// POUs/Remote/Objects/Basic/[Internal]/FB_BACnetRM_BaseObject
FUNCTION_BLOCK FB_BACnetRM_BaseObject IMPLEMENTS I_BACnetRM_BaseObject
VAR_INPUT CONSTANT
	{region 'Fixed Parameters'}
		{attribute 'parameterCategory':='General'}
		{attribute 'no_copy'}
		Client : REFERENCE TO FB_BACnet_Client;
		{attribute 'parameterCategory':='General'}
		nObjectInstance : UDINT := 16#003FFFFF;	
	{endregion}
END_VAR
VAR
	{region 'Output-Properties'}
		bReady				: BOOL;
	{endregion}
	{region 'SubInit'}
		eObjectType			: E_BACnetObjType				:= 16#FFFF;
		{attribute 'hide'}
		iOwner				: I_BACnetRM_ObjectOwner;												// Owner of current Instance (Pointer to current instance per default)
	{endregion}
END_VAR
VAR
	{region 'General'}
		eErrorID			: E_BACnet_Error				:= E_BACnet_Error.eNoError;
			 
		tObjectID			: T_BACnet_ObjectIdentifier		:= 16#FFFFFFFF;
	{endregion}
END_VAR

IF (NOT bReady) THEN
	IF (iOwner = 0) THEN
		eErrorID := E_BACnet_Error.eInvalidParameter;
		F_BA_LogMessage(ADSLOG_MSGTYPE_ERROR, 'O04', 'Owner of BACnet remote-object not defined!');
		
	ELSIF (__ISVALIDREF(Client)) THEN
		eErrorID := E_BACnet_Error.eNoError;
		bReady := TRUE;
		
		tObjectID := F_BACnet_GetObjId(eObjectType, nObjectInstance);
		
		OnObjectStateChanged();
		
		Client.UpdateRequests();
	ELSE
		eErrorID := E_BACnet_Error.eInvalidClient;
		iOwner.LogMsg.Show(ADSLOG_MSGTYPE_ERROR, 'O17', 'Assigned client-reference is invalid!', FALSE);
	END_IF
ELSE
	// Instance is operational.
END_IF

{attribute 'hide'}
METHOD OnCOV
VAR_INPUT
	ePropID		: E_BACnetPropIdentifier;
END_VAR
// Notify owner:
iOwner.OnBACnetRMObjectCOV(ePropID);
END_METHOD

{attribute 'hide'}
METHOD OnReqError
VAR_INPUT
	iRequest		: I_BACnetRM_Req;
	
	eResult			: E_BACnetRM_Error;
	sLogCode		: STRING			:= '';
END_VAR
VAR
	nLogType		: DWORD;
END_VAR

// (BETA) ... TODO
(*
... eResult ...

eErrorID := ;
nLogType := ADSLOG_MSGTYPE_ERROR;
nLogType := ADSLOG_MSGTYPE_WARN;
*)

iOwner.LogMsg.Show(nLogType, sLogCode, 'TODO: Implement request error!', FALSE);
END_METHOD

METHOD PROTECTED OnObjectStateChanged
// Notify owner:
iOwner.OnBACnetRMObjectStateChanged();
END_METHOD

PROPERTY Error : BOOL
GET
Error := (eErrorID <> E_BACnet_Error.eNoError);
END_GET
END_PROPERTY

PROPERTY ObjectID : T_BACnet_ObjectIdentifier
GET
ObjectID := tObjectID;
END_GET
END_PROPERTY

PROPERTY ObjectInstance : UDINT
GET
ObjectInstance := nObjectInstance;
END_GET
END_PROPERTY

PROPERTY ObjectType : E_BACnetObjType
GET
ObjectType := eObjectType;
END_GET
END_PROPERTY

PROPERTY Ready : BOOL
GET
Ready := bReady;
END_GET
END_PROPERTY

METHOD SyncProperty : BOOL
VAR_INPUT
	ePropID : E_BACnetPropIdentifier;
	nSize : UDINT;
	pData : PVOID;
	eSyncMode : E_BA_SyncModeRM;
END_VAR
CASE (eSyncMode) OF
	E_BA_SyncModeRM.eRead:
		SyncProperty := Client.AddReadProp(ePropID, THIS^, nSize, pData, 16#FFFFFFFF);
	
	E_BA_SyncModeRM.eWrite:
		SyncProperty := Client.AddWriteProp(ePropID, THIS^, nSize, pData, 0, 0, 16);

ELSE
	iOwner.LogMsg.Show1(ADSLOG_MSGTYPE_ERROR, 'SP09', 'Invalid Sync-Mode "%d"!', F_INT(eSyncMode), FALSE);
END_CASE
END_METHOD

METHOD SyncPropertyPrio : BOOL
VAR_INPUT
	ePropID : E_BACnetPropIdentifier;
	nSize : UDINT;
	pData : PVOID;
	pEnable : POINTER TO BOOL := 0;
	pNull : POINTER TO BOOL := 0;
	priority : UDINT := 16;
END_VAR
SyncPropertyPrio := Client.AddWriteProp(ePropID, THIS^, nSize, pData, pEnable, pNull, priority);
END_METHOD

END_FUNCTION_BLOCK

// TEST/TestPackage/CLIENT
PROGRAM CLIENT
VAR
	fbClient			: FB_BACnet_Client					:= (nDeviceInstance := 3637294(*, eReadMode := E_BACnet_CommMode.eCov*));
	
	AV01				: FB_BACnetRM_AV					:= (Client := fbClient, nObjectInstance:=111);
	AVDsp				: FB_BACnetRM_AV_Disp				:= (Client := fbClient, nObjectInstance:=10001);
	AVSp				: FB_BACnetRM_AV_Setp				:= (Client := fbClient, nObjectInstance:=10002);
	AI01				: FB_BACnetRM_AI					:= (Client := fbClient, nObjectInstance:=10000);
	AO01				: FB_BACnetRM_AO					:= (Client := fbClient, nObjectInstance:=10000);
	
	BV01				: FB_BACnetRM_BV					:= (Client := fbClient, nObjectInstance:=99);
	BVDsp				: FB_BACnetRM_BV_Disp				:= (Client := fbClient, nObjectInstance:=10001);
	BVSp				: FB_BACnetRM_BV_Setp				:= (Client := fbClient, nObjectInstance:=10002);
	BI01				: FB_BACnetRM_BI					:= (Client := fbClient, nObjectInstance:=10000);
	BO01				: FB_BACnetRM_BO					:= (Client := fbClient, nObjectInstance:=10000);
	
	MV01				: FB_BACnetRM_MV					:= (Client := fbClient, nObjectInstance:=99);
	MVDsp				: FB_BACnetRM_MV_Disp				:= (Client := fbClient, nObjectInstance:=10001);
	MVSp				: FB_BACnetRM_MV_Setp				:= (Client := fbClient, nObjectInstance:=10002);
	MI01				: FB_BACnetRM_MI					:= (Client := fbClient, nObjectInstance:=10000);
	MO01				: FB_BACnetRM_MO					:= (Client := fbClient, nObjectInstance:=10000);
	
	TLog				: FB_BACnetRM_TLog					:= (Client := fbClient, nObjectInstance:=10000);
	TLM					: FB_BACnetRM_TLM					:= (Client := fbClient, nObjectInstance:=10000);
	Cal01				: FB_BACnetRM_Cal					:= (Client := fbClient, nObjectInstance:=10000);
	SchedA				: FB_BACnetRM_SchedA				:= (Client := fbClient, nObjectInstance:=10000);
	SchedB				: FB_BACnetRM_SchedB				:= (Client := fbClient, nObjectInstance:=10001);
	SchedM				: FB_BACnetRM_SchedM				:= (Client := fbClient, nObjectInstance:=10002);
	Loop1				: FB_BACnetRM_Loop					:= (Client := fbClient, nObjectInstance:=10000);
	Loop2				: FB_BACnetRM_CnvLoop				:= (Client := fbClient, nObjectInstance:=10000);
	
	NC_AlmStd			: FB_BACnetRM_NC					:= (Client := fbClient, nObjectInstance:=11);
	
	Acc					: FB_BACnetRM_Acc					:= (Client := fbClient, nObjectInstance:=10000);
	PC					: FB_BACnetRM_PC					:= (Client := fbClient, nObjectInstance:=10000);
	Prog				: FB_BACnetRM_Prog					:= (Client := fbClient, nObjectInstance:=10000);
END_VAR
VAR
	diag : ST_BACnet_Diagnosis;
	scanRes : ARRAY [0..99] OF ST_BACnetRM_ScanResult;
	syncTime : ST_BA_DateTime;
	
	bDiag : BOOL;
	bScan : BOOL;
	bGet : BOOL;
	bSync : BOOL;
END_VAR

fbClient();

AV01();
AVDsp();
AVSp();
AI01();
AO01();

BV01();
BVDsp();
BVSp();
BI01();
BO01();

MV01();
MVDsp();
MVSp();
MI01();
MO01();

TLog();
TLM();
Cal01();
SchedA();
SchedB();
SchedM();
Loop1();
Loop2();

NC_AlmStd();

Acc();
PC();
Prog();

IF bDiag THEN
	fbClient.Adapter.GetDiagnosis(ADR(diag));
END_IF

IF bScan THEN	
	fbClient.Adapter.StartScan();
	bScan:=FALSE;
END_IF

IF bGet THEN
	fbClient.Adapter.GetScanResult(ADR(scanRes), 100);
	bGet:=FALSE;
END_IF

IF bSync THEN
	fbClient.Adapter.TimeSync(ADR(syncTime), TRUE);
	bSync:=FALSE;
END_IF

END_PROGRAM

// POUs/Remote/FB_BACnet_Client
FUNCTION_BLOCK FB_BACnet_Client IMPLEMENTS I_BACnetRM_Object
VAR_INPUT CONSTANT
	{region 'Fixed Parameters'}
		{attribute 'parameterCategory':='General'}
		{attribute 'no_copy'}
		Adapter	: REFERENCE TO FB_BACnet_Adapter := BACnet_Globals.DefaultAdapter;
		{attribute 'parameterCategory':='General'}
		nDeviceInstance : UDINT;
	{endregion}
END_VAR
VAR_INPUT CONSTANT PERSISTENT
	{region 'Variable Parameters'}
		{attribute 'parameterCategory':='Communication'}
		nMaxParallelRequests : UDINT := 1;
		{attribute 'parameterCategory':='Communication'}
		nRPMPropertiesPerRequest : UDINT := 80;
		{attribute 'parameterCategory':='Communication'}
		tCOVLifeTime : TIME := T#300S;	
		{attribute 'parameterCategory':='Communication'}
		eReadMode : E_BACnet_CommMode;
		{attribute 'parameterCategory':='Communication'}
		tReadCycleTime : TIME := T#5S;
		{attribute 'parameterCategory':='Communication'}
		tWriteCycleTime : TIME := T#5S;
	{endregion}
END_VAR
VAR_OUTPUT
	bReady					: BOOL;
	eErrorID				: E_BACnet_Error;
	nAdsPort 				: UINT;
	bConnected  			: BOOL;
END_VAR
VAR
	{region 'General'}
		tObjectID			: T_BACnet_ObjectIdentifier		:= 16#FFFFFFFF;
	{endregion}
END_VAR
VAR
	{region 'General'}
		eState				: E_BACnetRM_ClientState;
	
		stSupportedServices	: ST_BACnet_ServicesSupportedBits;
	{endregion}
	{region 'Request Lists'}
		{region 'Read'}
			{attribute 'hide'}
			stReadList 		: POINTER TO ST_BACnetRM_ReadEntry;
			{attribute 'hide'}
			nReadList		: UDINT := 0;
			{attribute 'hide'}
			nReadMax		: UDINT := 0;
		{endregion}
		{region 'Write'}
			{attribute 'hide'}
			stWriteList		: POINTER TO ST_BACnetRM_WriteEntry;
			{attribute 'hide'}
			nWriteList		: UDINT := 0;
			{attribute 'hide'}
			nWriteMax		: UDINT := 0;	
		{endregion}
	{endregion}
	{region 'Request Fifo'}
		{region 'Cyclic'}
			{attribute 'hide'}
			stReqList		: POINTER TO ST_BACnetRM_ReqPtr := 0;
			{attribute 'hide'}
			nReqList		: UDINT := 0;
			{attribute 'hide'}
			nCurReq			: UDINT := 0;
		{endregion}
		{region 'Acyclic / Dynamic'}
			{attribute 'hide'}
			fbReadFifo		: FB_BACnetRM_ReqFifo := (Client := THIS^);
			{attribute 'hide'}
			fbWriteFifo		: FB_BACnetRM_ReqFifo := (Client := THIS^);
		{endregion}
				  
		nOpenReq			: UDINT := 0;
		{attribute 'hide'}
		bUpdateReqs			: BOOL;
	{endregion}
		 
	{region 'Internal'}
		{attribute 'hide'}
		iServer				: ITcIoBACnetPlcServer;
		{attribute 'hide'}
		iClient				: ITcIoBACnetPlcClient;
		{attribute 'hide'}
		iDevice				: ITcIoBACnetPlcDevice;
		{attribute 'hide'}
		_bCreated			: BOOL;
		{attribute 'hide'}
		nUpdateCountAdp		: UDINT := 0;
			 
		{attribute 'hide'}
		fbRead				: FB_BACnetRM_ReadProperty := (Client:=THIS^);
		{attribute 'hide'}
		_ClientStatus		: WORD;
		{attribute 'hide'}
		_ClientControl		: WORD;
	{endregion}
END_VAR
VAR_TEMP
	n						: UDINT := 0;
END_VAR

IF __ISVALIDREF(Adapter) THEN
	IF Adapter._nUpdateCount = nUpdateCountAdp THEN
		Adapter();
	END_IF
	(* remind current number of update counter *)
	nUpdateCountAdp := Adapter._nUpdateCount;
	
	IF iDevice = 0 THEN
		iDevice := Adapter.Device;
	END_IF
END_IF

IF iClient = 0 THEN
	IF iDevice <> 0 THEN
		IF S_OK <> iDevice.GetClientById(nDeviceInstance, ADR(iServer)) THEN
			IF NOT _bCreated THEN
				IF S_OK = iDevice.CreateClient(nDeviceInstance) THEN
					_bCreated := TRUE;
				END_IF
			END_IF			
		ELSE
			iServer.GetAdsPort(ADR(nAdsPort));
			IF S_OK <> iServer.TcQueryInterface(TC_GLOBAL_IID_LIST.IID_ITcIoBACnetPlcClient, ADR(iClient)) THEN
				eErrorID := E_BACnet_Error.eInvalidClient;
			END_IF
		END_IF
	END_IF
END_IF

IF iClient <> 0 THEN
	iServer.UpdateDeviceStatus(ADR(_ClientControl), ADR(_ClientStatus));	
	IF Adapter.bEthernetLink THEN
		bConnected := NOT (SHR((_ClientStatus AND 16#FF00), 8) < 4);
	ELSE
		bConnected := FALSE;
	END_IF
	CASE eState OF
		E_BACnetRM_ClientState.eInit:
			IF bConnected THEN
				tObjectID := F_BACnet_GetObjId(ObjectType, nDeviceInstance);
		
				IF stSupportedServices.bSuppReadProperty THEN
					eState:=E_BACnetRM_ClientState.eCalcAuto;
				ELSE
					eState:=E_BACnetRM_ClientState.eReadSupportedServices;
				END_IF
			END_IF
		E_BACnetRM_ClientState.eReadSupportedServices:
			IF fbRead.bReady THEN
				IF eReadMode = E_BACnet_CommMode.eAuto OR eReadMode = E_BACnet_CommMode.eRpm THEN
					fbReadFifo.bRpm:=stSupportedServices.bSuppReadPropertyMultiple;
				END_IF
				eState:=E_BACnetRM_ClientState.eCalcAuto;
			ELSIF fbRead.bError THEN
				eState:=E_BACnetRM_ClientState.eError;
			ELSIF NOT fbRead.bBusy THEN
				fbRead(iObject:=THIS^, ePropID:=E_BACnetPropIdentifier.PropProtocolServicesSupported, nData:=SIZEOF(stSupportedServices), pData:=ADR(stSupportedServices), bExecute:=TRUE);
			END_IF
			fbReadFifo.ProcessReadFifo();
		E_BACnetRM_ClientState.eCalcAuto:
			IF nReadList > 0 OR nWriteList>0 THEN
				IF eReadMode = E_BACnet_CommMode.eAuto THEN
					IF nReadList > 300 AND stSupportedServices.bSuppReadPropertyMultiple THEN
						eReadMode := E_BACnet_CommMode.eRpm;
					ELSIF stSupportedServices.bSuppSubscribeCOV THEN
						eReadMode := E_BACnet_CommMode.eCov;
					ELSIF stSupportedServices.bSuppReadPropertyMultiple THEN
						eReadMode := E_BACnet_CommMode.eRpm;
					ELSE
						eReadMode := E_BACnet_CommMode.eRp;
					END_IF
				END_IF
				eState:=E_BACnetRM_ClientState.eCreateRequests;
			ELSE
				eState:=E_BACnetRM_ClientState.eCycle;
			END_IF
			eState:=E_BACnetRM_ClientState.eCreateRequests;
		E_BACnetRM_ClientState.eCreateRequests:
			IF CreateReqList() THEN
				bUpdateReqs := FALSE;
				eState:=E_BACnetRM_ClientState.eCycle;
			END_IF
		E_BACnetRM_ClientState.eCycle:
			IF bUpdateReqs THEN
				eState:=E_BACnetRM_ClientState.eReInit;
				bUpdateReqs := FALSE;
			ELSE
				bReady:=TRUE;
				
				// Work on acyclic / dynamic requests:
				fbReadFifo.ProcessReadFifo();
				fbWriteFifo.ProcessWriteFifo();
				
				// Work on cyclic requests:
				IF stReqList <> 0 THEN
					WHILE nOpenReq < nMaxParallelRequests AND n<nReqList DO								
						IF stReqList[nCurReq].pPtr <> 0 AND_THEN stReqList[nCurReq].fbBase^.IsReady() THEN
							IF stReqList[nCurReq].fbBase^.Send() THEN
								nOpenReq:=nOpenReq+1;
							END_IF
						END_IF
						n:=n+1;
						nCurReq:=(nCurReq+1) MOD nReqList;
					END_WHILE
				END_IF
			END_IF
			IF NOT bConnected THEN
				eState:=E_BACnetRM_ClientState.eReInit;
			END_IF
		E_BACnetRM_ClientState.eReInit:
			DeleteReqList();
			eState:=E_BACnetRM_ClientState.eInit;
		E_BACnetRM_ClientState.eError:
			// Todo: add 5 sec timer 
			eState:=E_BACnetRM_ClientState.eReInit;
	END_CASE
END_IF

{attribute 'hide'}
METHOD OnCOV
VAR_INPUT
	ePropID		: E_BACnetPropIdentifier;
END_VAR
END_METHOD

{attribute 'hide'}
METHOD OnReqError
VAR_INPUT
	iRequest		: I_BACnetRM_Req;
	
	eResult			: E_BACnetRM_Error;
	sLogCode		: STRING			:= '';
END_VAR
VAR
	nLogType		: DWORD;
END_VAR
END_METHOD

METHOD INTERNAL OnRequestComplete
IF nOpenReq > 0 THEN
	nOpenReq:=nOpenReq-1;
END_IF
END_METHOD

METHOD INTERNAL AddFifoReadReq : BOOL
VAR_INPUT
	pReq : POINTER TO FB_BACnetRM_ReadProperty;
END_VAR
VAR
	entry : ST_BACnetRM_FifoEntry;
END_VAR
entry.fbRead:=pReq;
AddFifoReadReq:=fbReadFifo.AddFifoReq(entry);
END_METHOD

METHOD INTERNAL AddFifoWriteReq : BOOL
VAR_INPUT
	pReq : POINTER TO FB_BACnetRM_WriteProperty;
END_VAR
VAR
	entry : ST_BACnetRM_FifoEntry;
END_VAR
entry.fbWrite:=pReq;
AddFifoWriteReq:=fbWriteFifo.AddFifoReq(entry);
END_METHOD

METHOD INTERNAL UpdateRequests 
VAR_INPUT
END_VAR
bUpdateReqs:=TRUE;
END_METHOD

METHOD PRIVATE CreateReadReq : I_BACnetRM_Req
VAR_INPUT
	eReadMode : E_BACnet_CommMode;
	stEntry : ST_BACnetRM_ReadEntry;
END_VAR
VAR
	stPtr : ST_BACnetRM_ReqPtr;
END_VAR
CASE eReadMode OF
	E_BACnet_CommMode.eCov:
		stPtr.fbCov:=__NEW(FB_BACnetRM_ReqCov);
		IF stPtr.fbCov <> 0 THEN
			stPtr.fbCov^(Client:=THIS^,iObject:=stEntry.iObject,  ePropID:=stEntry.ePropID, tLifetime:=tCOVLifeTime, pData:=stEntry.pData, nData:=stEntry.nData);
			stPtr.fbCov^.InitTimer();
		END_IF
		CreateReadReq:=stPtr.iReq;
		RETURN;
	E_BACnet_CommMode.eCovC:
		stPtr.fbCov:=__NEW(FB_BACnetRM_ReqCov);
		IF stPtr.fbCov <> 0 THEN
			stPtr.fbCov^(Client:=THIS^,iObject:=stEntry.iObject, bConfirmed:=TRUE, ePropID:=stEntry.ePropID, tLifetime:=tCOVLifeTime, pData:=stEntry.pData, nData:=stEntry.nData);
			stPtr.fbCov^.InitTimer();
		END_IF
		CreateReadReq:=stPtr.iReq;
		RETURN;
	E_BACnet_CommMode.eCovU:
		stPtr.fbCov:=__NEW(FB_BACnetRM_ReqCov);
		IF stPtr.fbCov <> 0 THEN
			stPtr.fbCov^(Client:=THIS^,iObject:=stEntry.iObject, bUnsubscribed:=TRUE, ePropID:=stEntry.ePropID, tLifetime:=tCOVLifeTime, pData:=stEntry.pData, nData:=stEntry.nData);
			stPtr.fbCov^.InitTimer();
		END_IF
		CreateReadReq:=stPtr.iReq;
		RETURN;
	E_BACnet_CommMode.eRp:
		stPtr.fbRead:=__NEW(FB_BACnetRM_ReqRead);
		IF stPtr.fbRead <> 0 THEN
			stPtr.fbRead^(Client:=THIS^,iObject:=stEntry.iObject, tCycleTime:=tReadCycleTime, ePropID:=stEntry.ePropID, pData:=stEntry.pData, nData:=stEntry.nData);
			stPtr.fbRead^.InitTimer();
		END_IF
		CreateReadReq:=stPtr.iReq;
		RETURN;
	E_BACnet_CommMode.eRpm:
		stPtr.fbRpm:=__NEW(FB_BACnetRM_ReqRpm);
		IF stPtr.fbRpm <> 0 THEN
			stPtr.fbRpm^(Client:=THIS^,iObject:=stEntry.iObject, tCycleTime:=tReadCycleTime);
			stPtr.fbRpm^.InitTimer();
		END_IF
		CreateReadReq:=stPtr.iReq;
		RETURN;
END_CASE
END_METHOD

METHOD PRIVATE CreateReqList : BOOL
VAR_INPUT
END_VAR
VAR
	i : UDINT;
	nReqs : UDINT;
	stPtr : ST_BACnetRM_ReqPtr;
	nReqsLeft : UDINT;
END_VAR
DeleteReqList();

IF eReadMode = E_BACnet_CommMode.eRpm THEN
	nReqs:=((nReadList+nRPMPropertiesPerRequest-1)/nRPMPropertiesPerRequest);
ELSE
	nReqs := nReadList;
END_IF

nReqs:=nReqs+nWriteList;

IF nReqs = 0 THEN
	RETURN;
END_IF

stReqList:=__NEW(POINTER TO ST_BACnetRM_ReqPtr, nReqs);

IF stReqList = 0 THEN
	RETURN;
END_IF

IF eReadMode = E_BACnet_CommMode.eRpm THEN
	nReqsLeft:=nReadList;
	WHILE nReqsLeft > 0 DO
		 stPtr.fbRpm:=__NEW(FB_BACnetRM_ReqRpm);
		 IF stPtr.fbRpm = 0 THEN
			 RETURN;
		 END_IF
		 stPtr.fbRpm^(Client:=THIS^, iObject:=stReadList[i].iObject, tCycleTime:=tReadCycleTime, pEntries:=ADR(stReadList[i]), nEntries:=MIN(nRPMPropertiesPerRequest, nReqsLeft));
		 stPtr.fbRpm^.InitTimer();
		 stPtr.fbRpm^.UpdateRequest();
		 nReqsLeft:=MIN(0, nReqsLeft-nRPMPropertiesPerRequest);
		 stReqList[nReqList]:=stPtr;
		 i:=i+MIN(0, nReqsLeft-nRPMPropertiesPerRequest);
		 nReqList:=nReqList+1;
	END_WHILE
	
ELSIF (nReadList > 0) THEN
	FOR i:=0 TO nReadList-1 DO
		stReqList[nReqList].iReq := CreateReadReq(eReadMode, stReadList[i]);
		IF stReqList[nReqList].pPtr = 0 THEN
			RETURN;
		END_IF
		nReqList:=nReqList+1;
	END_FOR
END_IF

IF eReadMode = E_BACnet_CommMode.eCov OR eReadMode = E_BACnet_CommMode.eCovC OR eReadMode = E_BACnet_CommMode.eCovU THEN
	OptimizeCOV();
END_IF

IF (nWriteList > 0) THEN
	FOR i:=0 TO nWriteList-1 DO
		stReqList[nReqList].fbWrite := __NEW(FB_BACnetRM_ReqWrite);
		IF stReqList[nReqList].pPtr = 0 THEN
			RETURN;
		END_IF
		
		stReqList[nReqList].fbWrite^(Client:=THIS^, iObject:=stWriteList[i].iObject, ePropID:=stWriteList[i].ePropID, tCycleTime:=tWriteCycleTime, pData:=stWriteList[i].pData, nData:=stWriteList[i].nData, pEnable:=stWriteList[i].pEnable, pNull:=stWriteList[i].pNull, fCOVIncrement:=stWriteList[i].fCOVIncrement, nPriority:=stWriteList[i].nPriority);
		stReqList[nReqList].fbWrite^.InitTimer();
		nReqList:=nReqList+1;
	END_FOR
END_IF

nCurReq := 0;
nOpenReq := 0;
CreateReqList:=TRUE;
END_METHOD

METHOD PRIVATE DeleteReqList
VAR_INPUT
END_VAR
VAR
	i : UDINT;
END_VAR
IF nReqList > 0 AND stReqList <> 0 THEN
	FOR i:=0 TO nReqList-1 DO
		IF stReqList[i].nByte <> 0 THEN
			CASE stReqList[i].iReq.GetRequestType() OF
				E_BACnetRM_RequestType.eRead:__DELETE(stReqList[i].fbRead);
				E_BACnetRM_RequestType.eReadPropertyMultiple:__DELETE(stReqList[i].fbRpm); 
				E_BACnetRM_RequestType.eWrite:__DELETE(stReqList[i].fbWrite);
				E_BACnetRM_RequestType.eWritePropertyMultiple:__DELETE(stReqList[i].fbWpm);
				E_BACnetRM_RequestType.eCOV_C:__DELETE(stReqList[i].fbCov);
				E_BACnetRM_RequestType.eCOV:__DELETE(stReqList[i].fbCov);
				E_BACnetRM_RequestType.eCOV_U:__DELETE(stReqList[i].fbCov);
			END_CASE
		END_IF
	END_FOR
	__DELETE(stReqList);
	stReqList:=0;
	nReqList:=0;
END_IF
END_METHOD

// Optimizes request count per object.
// > If a single object has more than one request, these multiple requests can be handled via a single RPM-request.
METHOD PRIVATE OptimizeCOV : BOOL
VAR
	i : UDINT;
	j : UDINT;
END_VAR
IF (nReadList > 0) THEN
	FOR i:=0 TO nReadList-1 DO
		IF stReqList[i].fbCov^.Master = 0 THEN
			FOR j:=i+1 TO nReadList-1 DO
				IF stReqList[i].fbCov^.iObject = stReqList[j].fbCov^.iObject THEN
					 stReqList[i].fbCov^.AddCovSlave(stReqList[j].fbCov);
					 stReqList[j].fbCov^.Master:=stReqList[i].fbCov;
					 IF stReqList[i].fbCov^.fCOVIncrement = 0 AND stReqList[i].fbCov^.ePropID = E_BACnetPropIdentifier.PropPresentValue AND stReqList[j].fbCov^.ePropID = E_BACnetPropIdentifier.PropStatusFlags THEN
						  stReqList[j].fbCov^.SendSubscription:=FALSE;
					 END_IF
				END_IF
			END_FOR
		END_IF
	END_FOR
END_IF
END_METHOD

// Called after online change.
{attribute 'call_after_online_change_slot' := '10'}
METHOD PROTECTED OnPostOnlineChange
IF iServer <> 0 THEN
	FW_SafeRelease(ADR(iServer));
	iServer:=0;
END_IF
IF iClient <> 0 THEN
	FW_SafeRelease(ADR(iClient));
	iClient:=0;
END_IF
iDevice:=0;

eState:=E_BACnetRM_ClientState.eReInit;
END_METHOD

METHOD FB_Exit : BOOL
VAR_INPUT
	 bInCopyCode : BOOL; // if TRUE, the exit method is called for exiting an instance that is copied afterwards (online change).
END_VAR
IF iServer <> 0 THEN
	iServer.OnPlcAction(E_BACnet_PlcAction.eSuspend);
	iServer:=0;
END_IF
IF iClient <> 0 THEN
	FW_SafeRelease(ADR(iClient));
	iClient:=0;
END_IF

iDevice:=0;

DeleteReqList();

IF stReadList <> 0 THEN
	__DELETE(stReadList);
	stReadList:=0;
END_IF
IF stWriteList <> 0 THEN
	__DELETE(stWriteList);
	stWriteList:=0;
END_IF
END_METHOD

PROPERTY Error : BOOL
GET
Error := (eErrorID <> E_BACnet_Error.eNoError);
END_GET
END_PROPERTY

PROPERTY ObjectID : T_BACnet_ObjectIdentifier
GET
ObjectID := tObjectID;
END_GET
END_PROPERTY

PROPERTY ObjectInstance : UDINT
GET
ObjectInstance := nDeviceInstance;
END_GET
END_PROPERTY

PROPERTY ObjectType : E_BACnetObjType
GET
ObjectType := E_BACnetObjType.ObjDevice;
END_GET
END_PROPERTY

PROPERTY OpenRequestCount : UDINT
GET
OpenRequestCount:=nOpenReq;
END_GET
SET
nOpenReq:=OpenRequestCount;
END_SET
END_PROPERTY

PROPERTY Ready : BOOL
GET
Ready := bReady;
END_GET
END_PROPERTY

METHOD AddReadProp : BOOL
VAR_INPUT
	ePropID : E_BACnetPropIdentifier;
	iObject : I_BACnetRM_BaseObject;
	nData : UDINT;
	pData : PVOID;
	nIndex : UDINT := 16#FFFFFFFF;
END_VAR
VAR
	nTmp : UDINT;
	nTmpSize : UDINT;
	pTmp : PVOID;
END_VAR
IF nReadList+1 >= nReadMax THEN
	nTmp := nReadMax+10;
	nTmpSize := nTmp*SIZEOF(ST_BACnetRM_ReadEntry);
	pTmp := __NEW(BYTE,nTmpSize);
	IF pTmp = 0 THEN
		RETURN;
	END_IF
	IF stReadList <> 0 THEN
		MEMCPY(pTmp, stReadList, nReadMax*SIZEOF(ST_BACnetRM_ReadEntry));
		__DELETE(stReadList);
	END_IF
	stReadList:=pTmp;
	nReadMax:=nTmp;
END_IF

MEMSET(ADR(stReadList[nReadList]), 0, SIZEOF(ST_BACnetRM_ReadEntry));

stReadList[nReadList].iObject:=iObject;
stReadList[nReadList].ePropID:=ePropID;
stReadList[nReadList].pData:=pData;
stReadList[nReadList].nData:=nData;
stReadList[nReadList].nIndex:=nIndex;

nReadList := nReadList + 1;

AddReadProp:=TRUE;
END_METHOD

METHOD AddWriteProp : BOOL
VAR_INPUT
	ePropID : E_BACnetPropIdentifier;
	iObject : I_BACnetRM_BaseObject;
	nData : UDINT;
	pData : PVOID;
	pEnable : POINTER TO BOOL := 0;
	pNull : POINTER TO BOOL := 0;
	nPriority : UDINT := 16;
END_VAR
VAR
	nTmp : UDINT;
	nTmpSize : UDINT;
	pTmp : PVOID;
END_VAR
IF nWriteList+1 >= nWriteMax THEN
	nTmp := nWriteMax+10;
	nTmpSize := nTmp*SIZEOF(ST_BACnetRM_WriteEntry);
	pTmp := __NEW(BYTE,nTmpSize);
	IF pTmp = 0 THEN
		RETURN;
	END_IF
	IF stWriteList <> 0 THEN
		MEMCPY(pTmp, stWriteList, nWriteMax*SIZEOF(ST_BACnetRM_WriteEntry));
		__DELETE(stWriteList);
	END_IF
	stWriteList:=pTmp;
	nWriteMax:=nTmp;
END_IF

MEMSET(ADR(stWriteList[nWriteList]), 0, SIZEOF(ST_BACnetRM_WriteEntry));

stWriteList[nWriteList].iObject:=iObject;
stWriteList[nWriteList].ePropID:=ePropID;
stWriteList[nWriteList].pData:=pData;
stWriteList[nWriteList].nData:=nData;
stWriteList[nWriteList].nPriority:=nPriority;
stWriteList[nWriteList].pEnable:=pEnable;
stWriteList[nWriteList].pNull:=pNull;
stWriteList[nWriteList].fCOVIncrement := 0.0;

nWriteList := nWriteList + 1;

AddWriteProp:=TRUE;
END_METHOD

END_FUNCTION_BLOCK

// POUs/Remote/Requests/[Internal]/FB_BACnetRM_ReqFifo
{attribute 'c++_compatible'}
{attribute 'enable_dynamic_creation'}
{attribute 'hide'}
FUNCTION_BLOCK FB_BACnetRM_ReqFifo EXTENDS FB_BACnetRM_ReqBase
VAR_INPUT
	bRpm : BOOL;
	bWpm : BOOL;
END_VAR
VAR
	pReqFifo	: POINTER TO ST_BACnetRM_FifoEntry;
	nReqFifo	: UDINT := 0;
	nMaxFifo	: UDINT := 0;
	nPendFifo	: UDINT := 0;
END_VAR

METHOD INTERNAL AddFifoReq : BOOL
VAR_INPUT
	pEntry : ST_BACnetRM_FifoEntry;
END_VAR
VAR
	nTmp : UDINT;
	nTmpSize : UDINT;
	pTmp : POINTER TO ST_BACnetRM_FifoEntry;
END_VAR
IF nReqFifo+1 >= nMaxFifo THEN
	nTmp := 2*nMaxFifo+100;
	nTmpSize := nTmp*SIZEOF(ST_BACnetRM_FifoEntry);
	pTmp := __NEW(BYTE,nTmpSize);
	IF pTmp = 0 THEN
		RETURN;
	END_IF
	IF pReqFifo <> 0 THEN
		MEMCPY(pTmp, pReqFifo, nMaxFifo*SIZEOF(ST_BACnetRM_FifoEntry));
		__DELETE(pReqFifo);
	END_IF
	pReqFifo:=pTmp;
	nMaxFifo:=nTmp;
END_IF

pReqFifo[nReqFifo]:=pEntry;
nReqFifo:=nReqFifo+1;

AddFifoReq:=TRUE;
END_METHOD

METHOD INTERNAL ProcessReadFifo : BOOL
VAR_INPUT
END_VAR
VAR
	pRequest : ST_BACnetRM_ReqPtr;
	nSize : UDINT;
	n :UDINT;
	pEntries : POINTER TO ST_BACnetRM_ReadEntry;
	
	x : UDINT;
END_VAR
IF IsValid THEN
	WHILE Client.nOpenReq < Client.nMaxParallelRequests AND nReqFifo > 0 DO		
		IF bRpm AND nReqFifo>1 THEN
			n:=0;
			nSize:=MIN(nReqFifo, Client.nRPMPropertiesPerRequest)*SIZEOF(ST_BACnetRM_ReadEntry);
			pRequest.fbRpm := __NEW(FB_BACnetRM_ReqRpm);
			IF pRequest.fbRpm = 0 THEN
				RETURN;
			END_IF
			pEntries:=__NEW(BYTE,nSize);
			IF pEntries = 0 THEN
				__DELETE(pRequest.fbRpm);
				RETURN;
			END_IF
			WHILE n<nReqFifo AND n < Client.nRPMPropertiesPerRequest DO
				pEntries[n].iObject:=pReqFifo[n].fbRead^.iObject;
				pEntries[n].ePropID:=pReqFifo[n].fbRead^.ePropID;
				pEntries[n].pData:=pReqFifo[n].fbRead^.pData;
				pEntries[n].nData:=pReqFifo[n].fbRead^.nData;
				pEntries[n].nIndex:=pReqFifo[n].fbRead^.nIndex;
				pEntries[n].fbReadProp:=pReqFifo[n].fbRead;
				n:=n+1;
			END_WHILE		
			pRequest.fbRpm^(Client:=Client, pEntries:=pEntries, nEntries:=n, bFreeEntries:=TRUE);
			IF pRequest.fbRpm^.UpdateRequest() AND_THEN pRequest.fbRpm^.Send() THEN
				Client.OpenRequestCount:=Client.nOpenReq+1;
				pReqFifo[0].fbRead^.Request:=pRequest;
				pReqFifo[0].fbRead^.bRequestRPM:=TRUE;
				MEMMOVE(pReqFifo, ADR(pReqFifo[n]), n*SIZEOF(ST_BACnetRM_ReadEntry));
				nReqFifo:=nReqFifo-n;
			ELSE
				__DELETE(pRequest.fbRpm);
				RETURN;
			END_IF
		ELSE
			pRequest.fbRead := __NEW(FB_BACnetRM_ReqRead);
			IF pRequest.fbRead = 0 THEN
				RETURN;
			END_IF
			pRequest.fbRead^(Client:=Client, iObject:=pReqFifo[0].fbRead^.iObject, pData:=pReqFifo[0].fbRead^.pData, nData:=pReqFifo[0].fbRead^.nData, ePropID:=pReqFifo[0].fbRead^.ePropID, fbReadProp:=pReqFifo[0].fbRead);
			IF pRequest.fbRead^.Send() THEN
				Client.OpenRequestCount:=Client.nOpenReq+1;
				pReqFifo[0].fbRead^.Request:=pRequest;	
				pReqFifo[0].fbRead^.bRequestRPM:=FALSE;
				MEMMOVE(pReqFifo, ADR(pReqFifo[1]), 1*SIZEOF(ST_BACnetRM_ReadEntry));
				nReqFifo:=nReqFifo-1;
			ELSE
				__DELETE(pRequest.fbRead);
				RETURN;
			END_IF
		END_IF
	END_WHILE
	
	ProcessReadFifo:=TRUE;
ELSE
	// (BETA) ... Output Error
END_IF
END_METHOD

METHOD INTERNAL ProcessWriteFifo : BOOL
VAR_INPUT
END_VAR
VAR
	pRequest : ST_BACnetRM_ReqPtr;
	nSize : UDINT;
	n :UDINT;
	pEntries : POINTER TO ST_BACnetRM_ReadEntry;
END_VAR
IF IsValid THEN
	WHILE Client.nOpenReq < Client.nMaxParallelRequests AND nReqFifo > 0 DO		
		IF bWpm THEN
			n:=0;
			nSize:=MIN(nReqFifo, Client.nRPMPropertiesPerRequest)*SIZEOF(ST_BACnetRM_ReadEntry);
			pRequest.fbWpm:= __NEW(FB_BACnetRM_ReqWpm);
			IF pRequest.fbWpm = 0 THEN
				RETURN;
			END_IF
			pEntries:=__NEW(BYTE,nSize);
			IF pEntries = 0 THEN
				__DELETE(pRequest.fbWpm);
				RETURN;
			END_IF
			WHILE n<nReqFifo-1 AND n < Client.nRPMPropertiesPerRequest DO
				pEntries[n].iObject:=pReqFifo[n].fbWrite^.iObject;
				pEntries[n].ePropID:=pReqFifo[n].fbWrite^.ePropID;
				pEntries[n].pData:=pReqFifo[n].fbWrite^.pData;
				pEntries[n].nData:=pReqFifo[n].fbWrite^.nData;
				pEntries[n].nIndex:=pReqFifo[n].fbWrite^.nIndex;
				pEntries[n].fbReadProp:=pReqFifo[n].fbWrite;
				n:=n+1;
			END_WHILE
			pRequest.fbWpm^(Client:=Client, pEntries:=pEntries, nEntries:=n, bFreeEntries:=TRUE);
			IF pRequest.fbWpm^.UpdateRequest() AND_THEN pRequest.fbWpm^.Send() THEN
				Client.OpenRequestCount:=Client.nOpenReq+1;
				pReqFifo[0].fbRead^.Request:=pRequest;
				pReqFifo[0].fbWrite^.bRequestWPM:=TRUE;
				MEMMOVE(pReqFifo, ADR(pReqFifo[n]), n*SIZEOF(ST_BACnetRM_ReadEntry));
				nReqFifo:=nReqFifo-n;
			ELSE
				__DELETE(pRequest.fbWpm);
				RETURN;
			END_IF
		ELSE
			pRequest.fbWrite := __NEW(FB_BACnetRM_ReqWrite);
			IF pRequest.fbWrite = 0 THEN
				RETURN;
			END_IF
			pRequest.fbWrite^(Client:=Client, iObject:=pReqFifo[0].fbWrite^.iObject, ePropID:=pReqFifo[0].fbWrite^.ePropID, pData:=pReqFifo[0].fbWrite^.pData, nData:=pReqFifo[0].fbWrite^.nData, fbWriteProp:=pReqFifo[0].fbWrite);
			IF pRequest.fbWrite^.Send() THEN
				pReqFifo[0].fbWrite^.Request:=pRequest;	
				pReqFifo[0].fbWrite^.bRequestWPM:=FALSE;
				Client.OpenRequestCount:=Client.nOpenReq+1;
				MEMMOVE(pReqFifo, ADR(pReqFifo[1]), 1*SIZEOF(ST_BACnetRM_ReadEntry));
			ELSE
				__DELETE(pRequest.fbWrite);
				RETURN;
			END_IF
		END_IF
	END_WHILE
	
	ProcessWriteFifo:=TRUE;
ELSE
	// (BETA) ... Output Error
END_IF
END_METHOD

METHOD FB_Exit : BOOL
VAR_INPUT
	 bInCopyCode : BOOL; // if TRUE, the exit method is called for exiting an instance that is copied afterwards (online change).
END_VAR
IF pReqFifo <> 0 THEN
	__DELETE(pReqFifo);
	pReqFifo:=0;
END_IF
END_METHOD

PROPERTY IsValid : BOOL
GET
// Hint:
// > Don't call "super()"!
//   The "iObject" Interface-pointer is ignored to this instance because it is unused.
IsValid := (__ISVALIDREF(Client));
END_GET
END_PROPERTY

END_FUNCTION_BLOCK

// POUs/Remote/Requests/[Internal]/[Base]/FB_BACnetRM_ReqBase
{attribute 'c++_compatible'}
{attribute 'enable_dynamic_creation'}
{attribute 'hide'}
FUNCTION_BLOCK FB_BACnetRM_ReqBase IMPLEMENTS I_BACnetRM_Req
VAR_INPUT
	{attribute 'initialize_on_call'}
	{attribute 'no_copy'}
	Client : REFERENCE TO FB_BACnet_Client;
	iObject : I_BACnetRM_BaseObject;
END_VAR

METHOD GetRequestType : E_BACnetRM_RequestType
VAR_INPUT
END_VAR
GetRequestType:=E_BACnetRM_RequestType.eUndefined;
END_METHOD

METHOD IsReady : BOOL
VAR_INPUT
END_VAR
END_METHOD

PROPERTY IsValid : BOOL
GET
VAR
	iTest : BOOL;
END_VAR
IsValid := (__ISVALIDREF(Client)) AND (iObject <> 0);
END_GET
END_PROPERTY

METHOD Send : BOOL
VAR
	_ClTmp : ITcIoBACnetPlcClient;
END_VAR
END_METHOD

END_FUNCTION_BLOCK

// POUs/Remote/Requests/[Internal]/FB_BACnetRM_ReqRpm
{attribute 'c++_compatible'}
{attribute 'enable_dynamic_creation'}
{attribute 'hide'}
FUNCTION_BLOCK FB_BACnetRM_ReqRpm EXTENDS FB_BACnetRM_ReqBasic
VAR_INPUT
	pEntries : POINTER TO ST_BACnetRM_ReadEntry;
	nEntries : UDINT;
	bFreeEntries : BOOL; 
END_VAR
VAR_OUTPUT
	bInit : BOOL;
END_VAR
VAR 
	req : SendDataRequest;
	pTmp : POINTER TO ST_BACnetRM_RpmListEntry;
END_VAR

IF NOT __ISVALIDREF(Client) THEN
	bError:=TRUE;
END_IF

SUPER^();

{attribute 'hide'}
METHOD Send : BOOL
IF IsValid THEN
	IF stReq = 0 THEN
		RETURN;
	END_IF
	
	Send:=SUPER^.Send();
ELSE
	// (BETA) ... Output Error
END_IF
END_METHOD

METHOD INTERNAL UpdateRequest : BOOL
VAR_INPUT
END_VAR
VAR
	nSize : UDINT;
	i : UDINT;
	nTmpSize : UDINT;
END_VAR
IF IsValid THEN
	IF stReq <> 0 AND_THEN stReq^.pData <> 0 THEN
		pTmp:=stReq^.pData;
		__DELETE(pTmp);
		stReq^.pData:=0;
	END_IF
	nTmpSize := SIZEOF(ST_BACnetRM_RpmListEntry)*nEntries;
	pTmp := __NEW(BYTE,nTmpSize);
	IF pTmp = 0 THEN
		RETURN;
	END_IF
	
	FOR i:=0 TO nEntries-1 DO
		pTmp[i].tObjectID := pEntries[i].iObject.ObjectID;
		pTmp[i].ePropID := pEntries[i].ePropID;
		pTmp[i].nArrayIndex := 0;
		pTmp[i].nValidBits := 0;
		pTmp[i].nPriority := 0;
		pTmp[i].nEntrySize := SIZEOF(ST_BACnetRM_RpmListEntry) - 8;
		IF i <> nEntries -1 THEN
			pTmp[i].nEntrySize := pTmp[i].nEntrySize + 16#80000000;
		END_IF
	END_FOR
	
	stReq := ADR(req);
	stReq^.pData := pTmp;
	stReq^.nData := nTmpSize;
	
	stReq^.service := E_BACnetConfirmedService.SrvReadPropertyMultiple;
	stReq^.deviceId := Client.ObjectInstance;
	
	bInit:=TRUE;
	
	UpdateRequest:=TRUE;
ELSE
	// (BETA) ... Output Error
END_IF
END_METHOD

METHOD PRIVATE Free
VAR_INPUT
END_VAR
IF bFreeEntries AND pEntries <> 0 THEN
	__DELETE(pEntries);
	pEntries:=0;
	bFreeEntries:=FALSE;
END_IF

IF stReq <> 0 AND_THEN stReq^.pData <> 0 THEN
	pTmp:=req.pData;
	__DELETE(pTmp);
	req.pData:=0;
	stReq:=0;
END_IF
END_METHOD

METHOD PROTECTED OnError
VAR_INPUT
	eResult			: E_BACnetRM_Error;
	sLogCode		: STRING			:= '';
END_VAR
VAR
	i : UDINT;
END_VAR
// Do not call super! Handle each entry's error:
// SUPER^.OnError(eResult, sLogCode);

FOR i:=0 TO nEntries-1 DO
	IF pEntries[i].fbReadProp <> 0 THEN
		pEntries[i].fbReadProp^.Busy:=FALSE;
		pEntries[i].fbReadProp^.Error:=TRUE;

		IF (pEntries[i].iObject <> 0) THEN
			pEntries[i].iObject.OnReqError(THIS^, E_BACnetRM_Error.eKillMe, 'OE07');
		END_IF	
	END_IF
END_FOR
END_METHOD

METHOD PROTECTED ProcessResult : HRESULT
VAR_INPUT
	pResult	: POINTER TO SendDataRequestResult;
END_VAR
VAR
	pPropList : POINTER TO ST_BACnetRM_RpmListEntry;
	i : UDINT;
END_VAR
IF pResult^.service <> E_BACnetConfirmedService.SrvReadPropertyMultiple THEN
	OnError(E_BACnetRM_Error.eInvalidService,  '');
	bError:=TRUE;
	RETURN;
END_IF

// set all entries to error, all good entries in response will be set to good afterwards
FOR i:=0 TO nEntries-1 DO
	IF pEntries[i].fbReadProp <> 0 THEN
		pEntries[i].fbReadProp^.Ready:=FALSE;	
		pEntries[i].fbReadProp^.Busy:=FALSE;
		pEntries[i].fbReadProp^.Error:=TRUE;
	END_IF
	
	pEntries[i]._bError := TRUE;
END_FOR

// copy data:
pPropList := pResult^.pData;
WHILE pPropList <> 0 DO
	_WritePropEntry(pPropList);
	pPropList := F_BACnet_NextListElem(pPropList, pPropList^.nEntrySize);
	bReady:=TRUE;
END_WHILE

// Evaluate remaining errors:
FOR i:=0 TO nEntries-1 DO
	IF (pEntries[i]._bError) AND_THEN (pEntries[i].iObject <> 0) THEN
		pEntries[i].iObject.OnReqError(THIS^, E_BACnetRM_Error.eKillMe, 'OE28');
	END_IF
END_FOR
END_METHOD

METHOD PRIVATE _WritePropEntry : BOOL
VAR_INPUT
	pEntry : POINTER TO ST_BACnetRM_RpmListEntry;
END_VAR
VAR
	i : UDINT;
END_VAR
FOR i:=0 TO nEntries-1 DO
	IF (pEntries[i].iObject.ObjectID = pEntry^.tObjectID) AND (pEntries[i].ePropID = pEntry^.ePropID) THEN
		CopyRemoteData(pEntries[i].iObject, pEntry^.ePropID ,pEntries[i].pData, pEntries[i].nData, F_BACnet_EndOf(pEntry, SIZEOF(ST_BACnetRM_RpmListEntry)), pEntry^.nEntrySize-16); 
		IF pEntries[i].fbReadProp <> 0 THEN
			pEntries[i].fbReadProp^.Ready:=TRUE;	
			pEntries[i].fbReadProp^.Busy:=FALSE;
			pEntries[i].fbReadProp^.Error:=FALSE;
		END_IF
		pEntries[i]._bError := FALSE;
		
		_WritePropEntry:=TRUE;
	END_IF
END_FOR
END_METHOD

METHOD FB_exit : BOOL
VAR_INPUT
	bInCopyCode : BOOL; // if TRUE, the exit method is called for exiting an instance that is copied afterwards (online change).
END_VAR
Free();
END_METHOD

METHOD GetRequestType : E_BACnetRM_RequestType
VAR_INPUT
END_VAR
GetRequestType := E_BACnetRM_RequestType.eReadPropertyMultiple;
END_METHOD

END_FUNCTION_BLOCK

// POUs/Remote/Requests/[Internal]/[Base]/FB_BACnetRM_ReqBasic
{attribute 'c++_compatible'}
{attribute 'enable_dynamic_creation'}
{attribute 'hide'}
FUNCTION_BLOCK FB_BACnetRM_ReqBasic EXTENDS FB_BACnetRM_ReqBase IMPLEMENTS ITcIoBACnetServiceResponseSink
VAR_INPUT
	tCycleTime : TIME := T#5S;
END_VAR
VAR_OUTPUT
	bBusy : BOOL;
	bError : BOOL;
	bReady : BOOL;
END_VAR
VAR
	{attribute 'hide'}
	stReq : POINTER TO SendDataRequest;
	timer : TON;
END_VAR

{attribute 'c++_compatible'}
{attribute 'minimal_input_size' := '4'}
{attribute 'pack_mode' := '4'}
{attribute 'hide'}
METHOD OnSendPropertyDataRequest : HRESULT
VAR_INPUT
	pResult	: POINTER TO SendDataRequestResult;
END_VAR
IF IsValid THEN
	IF pResult <> 0 THEN
		IF F_BACnetRM_IsErrorSet(pResult) THEN
			bBusy := FALSE;
			bError := TRUE;
			OnError(E_BACnetRM_Error.eKillMe, 'OE08');
			OnSendPropertyDataRequest:=S_FALSE;
		ELSE
			bError := FALSE;
			OnSendPropertyDataRequest:=ProcessResult(pResult);
			bBusy := FALSE;
		END_IF
		Client.OnRequestComplete();
	END_IF
ELSE
	// (BETA) ... Output Error
END_IF
END_METHOD

METHOD INTERNAL InitTimer : BOOL
VAR_INPUT
END_VAR
timer(IN:=FALSE, PT:=T#1MS);
timer(IN:=TRUE, PT:=T#1MS);
END_METHOD

{attribute 'c++_compatible'}
{attribute 'minimal_input_size' := '4'}
{attribute 'pack_mode' := '4'}
{attribute 'hide'}
METHOD TcAddRef : UDINT
END_METHOD

{attribute 'c++_compatible'}
{attribute 'minimal_input_size' := '4'}
{attribute 'pack_mode' := '4'}
{attribute 'hide'}
METHOD TcQueryInterface : HRESULT
VAR_INPUT
	iid	: REFERENCE TO IID;
	pipItf	: POINTER TO PVOID;
END_VAR
VAR
	ipSink : ITcIoBACnetServiceResponseSink;
	ipUnknown : ITcUnknown;	
END_VAR
IF GuidsEqual(ADR(iid), ADR(TC_GLOBAL_IID_LIST.IID_ITcIoBACnetServiceResponseSink)) THEN
	ipSink := THIS^; // cast to interface pointer
	pipItf^ := ITCUNKNOWN_TO_PVOID(ipSink);
	TcAddRef();
	TcQueryInterface := S_OK;
ELSIF GuidsEqual(ADR(iid), ADR(TC_GLOBAL_IID_LIST.IID_ITcUnknown)) THEN
	ipUnknown := THIS^; // cast to interface pointer
	pipItf^ := ITCUNKNOWN_TO_PVOID(ipUnknown);
	TcAddRef();
	TcQueryInterface := S_OK;
ELSE
	TcQueryInterface := E_HRESULTAdsErr.NOINTERFACE ; //Call super if this fb extends some other
END_IF
END_METHOD

{attribute 'c++_compatible'}
{attribute 'minimal_input_size' := '4'}
{attribute 'pack_mode' := '4'}
{attribute 'hide'}
METHOD TcRelease : UDINT
END_METHOD

METHOD PROTECTED OnError
VAR_INPUT
	eResult			: E_BACnetRM_Error;
	sLogCode		: STRING			:= '';
END_VAR
IF (iObject <> 0) THEN
	iObject.OnReqError(THIS^, eResult, sLogCode);
END_IF
END_METHOD

METHOD PROTECTED CopyRemoteData : BOOL
VAR_INPUT
	iObject : I_BACnetRM_BaseObject;
	ePropID : E_BACnetPropIdentifier;
	pDst : PVOID;
	nDst : UDINT;
	pSrc : PVOID;
	nSrc : UDINT;
END_VAR
VAR
	i 	 : INT;
	pByte : POINTER TO BYTE;
	pSchedPv : POINTER TO ST_BACnet_ValueList;
END_VAR
CASE ePropID OF
	E_BACnetPropIdentifier.PropStatusFlags:
		pByte:=pDst;
		FOR i:=0 TO 3 DO
			IF F_BACnet_IsBitFieldBitSetPtr(pSrc, i) THEN
				pByte[i]:=1;
			ELSE
				pByte[i]:=0;
			END_IF
		END_FOR
	E_BACnetPropIdentifier.PropAckedTransitions:
		pByte:=pDst;
		FOR i:=0 TO 2 DO
			IF F_BACnet_IsBitFieldBitSetPtr(pSrc, i) THEN
				pByte[i]:=1;
			ELSE
				pByte[i]:=0;
			END_IF
		END_FOR
	E_BACnetPropIdentifier.PropEventEnable:
		pByte:=pDst;
		FOR i:=0 TO 2 DO
			IF F_BACnet_IsBitFieldBitSetPtr(pSrc, i) THEN
				pByte[i]:=1;
			ELSE
				pByte[i]:=0;
			END_IF
		END_FOR
	E_BACnetPropIdentifier.PropPresentValue:
		IF iObject.ObjectType = E_BACnetObjType.ObjSchedule THEN
			IF nSrc >= 16 THEN
				pSchedPv := pSrc;
				CASE pSchedPv^.listEntry.eValueChoice OF
					E_BACnet_ValueChoice.eBoolValue:
						MEMCPY(pDst, ADR(pSchedPv^.listEntry.stValue), MIN(SIZEOF(BOOL),nDst)); 
					E_BACnet_ValueChoice.eRealValue:
						MEMCPY(pDst, ADR(pSchedPv^.listEntry.stValue), MIN(SIZEOF(REAL),nDst)); 
					E_BACnet_ValueChoice.eUnsignedValue:
						MEMCPY(pDst, ADR(pSchedPv^.listEntry.stValue), MIN(SIZEOF(UDINT),nDst)); 
					E_BACnet_ValueChoice.eEnumerationValue:
						MEMCPY(pDst, ADR(pSchedPv^.listEntry.stValue.enumValue), MIN(SIZEOF(UDINT),nDst)); 
				END_CASE
			END_IF
		ELSE
			MEMCPY(pDst, pSrc, MIN(nSrc,nDst)); 
		END_IF
ELSE
	MEMCPY(pDst, pSrc, MIN(nSrc,nDst)); 
END_CASE

// Notify object about changed value:
iObject.OnCOV(ePropID);
END_METHOD

METHOD PROTECTED ProcessResult : HRESULT
VAR_INPUT
	pResult	: POINTER TO SendDataRequestResult;
END_VAR
ProcessResult:=S_OK;
END_METHOD

METHOD Send : BOOL
VAR
	_ClTmp : ITcIoBACnetPlcClient;
END_VAR
IF IsValid THEN
	_ClTmp := Client.iClient;
	
	IF S_OK = _ClTmp.SendPropertyDataRequest(stReq, THIS^) THEN
		Send:=TRUE;
		bBusy:=TRUE;
		StartTimer();
	ELSE
		Send:=FALSE; 
	END_IF
ELSE
	// (BETA) ... Output Error
END_IF
END_METHOD

METHOD PROTECTED StartTimer : BOOL
VAR_INPUT
END_VAR
timer(IN:=FALSE, PT:=tCycleTime);
timer(IN:=TRUE, PT:=tCycleTime);
END_METHOD

METHOD GetRequestType : E_BACnetRM_RequestType
VAR_INPUT
END_VAR
GetRequestType:=E_BACnetRM_RequestType.eUndefined;
END_METHOD

METHOD IsReady : BOOL
VAR_INPUT
END_VAR
timer(Q=>IsReady);
IF bBusy THEN
	IsReady:=FALSE;
END_IF
END_METHOD

END_FUNCTION_BLOCK

// POUs/Remote/Requests/[Internal]/FB_BACnetRM_ReqRead
{attribute 'c++_compatible'}
{attribute 'enable_dynamic_creation'}
{attribute 'hide'}
FUNCTION_BLOCK FB_BACnetRM_ReqRead EXTENDS FB_BACnetRM_ReqBasic
VAR_INPUT
	ePropID : E_BACnetPropIdentifier;
	pData : PVOID;
	nData : UDINT;
	fbReadProp : POINTER TO FB_BACnetRM_ReadProperty := 0;
END_VAR
VAR 
	req : SendDataRequest;
END_VAR

IF NOT __ISVALIDREF(Client) THEN
	bError:=TRUE;
END_IF

SUPER^();

{attribute 'hide'}
METHOD Send : BOOL
IF IsValid THEN
	IF stReq = 0 THEN
		IF ePropID = E_BACnetPropIdentifier.PropLogBuffer THEN
			req.service := E_BACnetConfirmedService.SrvReadRange;
		ELSE
			req.service := E_BACnetConfirmedService.SrvReadProperty;
		END_IF	
		req.objectIdentifier := iObject.ObjectID;
		req.propertyIdentifier := ePropID;
		req.pData := pData;
		req.nData := nData;
		req.deviceId := Client.ObjectInstance;
		stReq := ADR(req);
	END_IF
	
	Send:=SUPER^.Send();
ELSE
	// (BETA) ... Output Error
END_IF
END_METHOD

METHOD PROTECTED OnError
VAR_INPUT
	eResult			: E_BACnetRM_Error;
	sLogCode		: STRING			:= '';
END_VAR
SUPER^.OnError(eResult, sLogCode);

IF fbReadProp <> 0 THEN
	fbReadProp^.Busy:=FALSE;
	fbReadProp^.Error:=TRUE;
END_IF
END_METHOD

METHOD PROTECTED ProcessResult : HRESULT
VAR_INPUT
	pResult	: POINTER TO SendDataRequestResult;
END_VAR
IF IsValid THEN
	IF  pResult^.nData <= nData THEN
		CopyRemoteData(iObject, ePropID, pData, nData, pResult^.pData, pResult^.nData);
		bReady:=TRUE;
	ELSE
		bError:=TRUE;
	END_IF
	
	IF fbReadProp <> 0 THEN
		fbReadProp^.Busy:=FALSE;
		fbReadProp^.Ready:=TRUE;
	END_IF
ELSE
	// (BETA) ... Output Error
END_IF
END_METHOD

METHOD GetRequestType : E_BACnetRM_RequestType
VAR_INPUT
END_VAR
GetRequestType:=E_BACnetRM_RequestType.eRead;
END_METHOD

END_FUNCTION_BLOCK

// POUs/Remote/Requests/FB_BACnetRM_ReadProperty
FUNCTION_BLOCK FB_BACnetRM_ReadProperty EXTENDS FB_BACnetRM_BaseProperty
VAR_INPUT CONSTANT
	{attribute 'initialize_on_call'}
	{attribute 'no_copy'}
	Client : REFERENCE TO FB_BACnet_Client;
	
	bRequestRPM : BOOL;
END_VAR

IF bExecuteOld <> bExecute AND NOT bBusy THEN
	IF NOT IsValid THEN
		bError:=TRUE;
		bReady:=FALSE;
	END_IF
	bExecuteOld := bExecute;
	Free();
	
	IF NOT Client.AddFifoReadReq(THIS) THEN
		bError:=TRUE;
		bReady:=FALSE;
	ELSE
		bBusy:=TRUE;
		bError:=FALSE;
		bReady:=FALSE;
	END_IF
END_IF

METHOD PROTECTED OnExecuteChange : BOOL
OnExecuteChange := Client.AddFifoReadReq(THIS);
END_METHOD

METHOD PROTECTED Free : BOOL
IF pRequest.pPtr <> 0 THEN
	IF bRequestRPM THEN
		__DELETE(pRequest.fbRpm);
	ELSE
		__DELETE(pRequest.fbRead);
	END_IF
	pRequest.pPtr:=0;
END_IF
END_METHOD

METHOD FB_exit : BOOL
VAR_INPUT
	bInCopyCode : BOOL; // if TRUE, the exit method is called for exiting an instance that is copied afterwards (online change).
END_VAR
Free();
END_METHOD

PROPERTY IsValid : BOOL
GET
IsValid := __ISVALIDREF(Client);
END_GET
END_PROPERTY

END_FUNCTION_BLOCK

// POUs/Remote/Requests/[Internal]/[Base]/FB_BACnetRM_BaseProperty
FUNCTION_BLOCK FB_BACnetRM_BaseProperty
VAR_INPUT CONSTANT
	pData : PVOID;
	nData : UDINT;
	iObject : I_BACnetRM_BaseObject;
	nIndex : UDINT := 16;
	ePropID : E_BACnetPropIdentifier;
	bExecute : BOOL;
	{attribute 'hide'}
	pRequest : ST_BACnetRM_ReqPtr;
END_VAR
VAR_OUTPUT
	bReady : BOOL;
	bBusy : BOOL;
	bError : BOOL;
END_VAR
VAR
	{attribute 'hide'}
	bExecuteOld : BOOL;
END_VAR

IF bExecuteOld <> bExecute AND NOT bBusy THEN
	bError := NOT IsValid;
	bReady := FALSE;
	bExecuteOld := bExecute;
	
	Free();
	
	IF OnExecuteChange() THEN
		bBusy:=TRUE;
		bError:=FALSE;
	ELSE
		bError:=TRUE;
	END_IF
END_IF

METHOD PROTECTED OnExecuteChange : BOOL
OnExecuteChange := FALSE;
END_METHOD

METHOD PROTECTED Free : BOOL
Free := FALSE;
END_METHOD

PROPERTY Busy : BOOL
GET
Busy:=bBusy;
END_GET
SET
bBusy:=Busy;
END_SET
END_PROPERTY

PROPERTY Error : BOOL
GET
Error:=bError;
END_GET
SET
bError:=Error;
END_SET
END_PROPERTY

PROPERTY IsValid : BOOL
GET
IsValid := FALSE;
END_GET
END_PROPERTY

PROPERTY Ready : BOOL
GET
Ready:=bReady;
END_GET
SET
bReady:=Ready;
END_SET
END_PROPERTY

PROPERTY Request : ST_BACnetRM_ReqPtr;
GET
Request:=pRequest;
END_GET
SET
pRequest:=Request;
END_SET
END_PROPERTY

END_FUNCTION_BLOCK

// POUs/Remote/Requests/[Internal]/FB_BACnetRM_ReqWpm
{attribute 'c++_compatible'}
{attribute 'enable_dynamic_creation'}
{attribute 'hide'}
FUNCTION_BLOCK FB_BACnetRM_ReqWpm EXTENDS FB_BACnetRM_ReqBasic
VAR_INPUT
	pEntries : POINTER TO ST_BACnetRM_ReadEntry;
	nEntries : UDINT;
	bFreeEntries : BOOL; 
END_VAR
VAR_OUTPUT
	bInit : BOOL;
END_VAR
VAR 
	{attribute 'hide'}
	req : SendDataRequest;
	{attribute 'hide'}
	pTmp : POINTER TO ST_BACnetRM_RpmListEntry;
END_VAR

IF NOT __ISVALIDREF(Client) THEN
	bError:=TRUE;
END_IF

SUPER^();

{attribute 'hide'}
METHOD Send : BOOL
IF IsValid THEN
	IF stReq = 0 THEN
		Send:=FALSE;
		RETURN;
	END_IF
	
	UpdateRequest();
	Send:=SUPER^.Send();
ELSE
	// (BETA) ... Output Error
END_IF
END_METHOD

METHOD INTERNAL UpdateRequest : BOOL
VAR_INPUT
END_VAR
VAR
	nSize : UDINT;
	i : UDINT;
	nTmpSize : UDINT;
END_VAR
IF IsValid THEN
	IF stReq <> 0 AND_THEN stReq^.pData <> 0 THEN
		pTmp:=stReq^.pData;
		__DELETE(pTmp);
	END_IF
	FOR i:=0 TO nEntries-1 DO
		nTmpSize := nTmpSize + SIZEOF(ST_BACnetRM_RpmListEntry) + F_BACnet_AlignedSize(pEntries[i].nData);
	END_FOR
	pTmp := __NEW(BYTE,nTmpSize);
	IF pTmp = 0 THEN
		UpdateRequest:=FALSE;
		RETURN;
	END_IF
	
	stReq := ADR(req);
	stReq^.pData := pTmp;
	FOR i:=0 TO nEntries-1 DO
		pTmp^.tObjectID := pEntries[i].iObject.ObjectID;
		pTmp^.ePropID := pEntries[i].ePropID;
		pTmp^.nArrayIndex := 0;
		pTmp^.nValidBits := 0;
		pTmp^.nPriority := 0;
		pTmp^.nEntrySize := F_BACnet_AlignedSize(pEntries[i].nData) + SIZEOF(ST_BACnetRM_RpmListEntry) - 8;
		MEMCPY(F_BACnet_EndOf(pTmp, SIZEOF(ST_BACnetRM_RpmListEntry)), pEntries[i].pData, pEntries[i].nData); 
		IF i <> nEntries -1 THEN
			pTmp[i].nEntrySize := pTmp[i].nEntrySize + 16#80000000;
		END_IF
		pTmp := F_BACnet_NextListElem(pTmp, pTmp^.nEntrySize);
	END_FOR
	
	stReq^.nData := nTmpSize;
	stReq^.service := E_BACnetConfirmedService.SrvWritePropertyMultiple;
	stReq^.deviceId := Client.ObjectInstance;
	
	bInit:=TRUE;
	
	UpdateRequest:=TRUE;
ELSE
	// (BETA) ... Output Error
END_IF
END_METHOD

METHOD PRIVATE Free
VAR_INPUT
END_VAR
IF bFreeEntries AND pEntries <> 0 THEN
	__DELETE(pEntries);
	pEntries:=0;
	bFreeEntries:=FALSE;
END_IF

IF stReq <> 0 AND_THEN stReq^.pData <> 0 THEN
	pTmp:=req.pData;
	__DELETE(pTmp);
	req.pData:=0;
	stReq:=0;
END_IF
END_METHOD

METHOD PROTECTED OnError
VAR_INPUT
	eResult			: E_BACnetRM_Error;
	sLogCode		: STRING			:= '';
END_VAR
VAR
	i : UDINT;
END_VAR
// Do not call super! Handle each entry's error:
// SUPER^.OnError(eResult, sLogCode);

FOR i:=0 TO nEntries-1 DO
	IF pEntries[i].fbReadProp <> 0 THEN
		pEntries[i].fbReadProp^.Busy:=FALSE;
		pEntries[i].fbReadProp^.Error:=TRUE;	

		IF (pEntries[i].iObject <> 0) THEN
			pEntries[i].iObject.OnReqError(THIS^, E_BACnetRM_Error.eKillMe, 'OE10');
		END_IF		
	END_IF
END_FOR
END_METHOD

METHOD PROTECTED ProcessResult : HRESULT
VAR_INPUT
	pResult	: POINTER TO SendDataRequestResult;
END_VAR
VAR
	pPropList : POINTER TO ST_BACnetRM_RpmListEntry;
END_VAR
VAR
	i : UDINT;
END_VAR
IF pResult^.service <> E_BACnetConfirmedService.SrvWritePropertyMultiple THEN
	bError:=TRUE;
	RETURN;
END_IF

FOR i:=0 TO nEntries-1 DO
	IF pEntries[i].fbReadProp <> 0 THEN
			pEntries[i].fbReadProp^.Ready:=TRUE;	// TODO: handle error entry		
			pEntries[i].fbReadProp^.Busy:=FALSE;
	END_IF
END_FOR
bReady:=TRUE;
END_METHOD

METHOD FB_exit : BOOL
VAR_INPUT
	bInCopyCode : BOOL; // if TRUE, the exit method is called for exiting an instance that is copied afterwards (online change).
END_VAR
Free();
END_METHOD

METHOD GetRequestType : E_BACnetRM_RequestType
VAR_INPUT
END_VAR
GetRequestType := E_BACnetRM_RequestType.eWritePropertyMultiple;
END_METHOD

END_FUNCTION_BLOCK

// POUs/Remote/Requests/[Internal]/FB_BACnetRM_ReqWrite
{attribute 'c++_compatible'}
{attribute 'enable_dynamic_creation'}
{attribute 'hide'}
FUNCTION_BLOCK FB_BACnetRM_ReqWrite EXTENDS FB_BACnetRM_ReqBasic
VAR_INPUT CONSTANT
	ePropID : E_BACnetPropIdentifier;
	pData : PVOID;
	nData : UDINT;
	pEnable : POINTER TO BOOL;
	pNull : POINTER TO BOOL;
	fCOVIncrement : REAL;
	nPriority : UDINT := 16;
	{attribute 'hide'}
	fbWriteProp : POINTER TO FB_BACnetRM_WriteProperty;
END_VAR
VAR 
	{attribute 'hide'}
	req : SendDataRequest;
	{attribute 'hide'}
	lastWriteValue : ST_BACnetRM_LastWriteValue;
END_VAR

IF NOT __ISVALIDREF(Client) THEN
	bError:=TRUE;
END_IF

SUPER^();

{attribute 'hide'}
METHOD Send : BOOL
IF IsValid THEN
	IF stReq = 0 THEN
		req.service := E_BACnetConfirmedService.SrvWriteProperty;
		req.objectIdentifier := iObject.ObjectID;
		req.propertyIdentifier := ePropID;
		IF (F_BACnet_IsPriorityValid(TO_INT(nPriority))) THEN
			req.priority := nPriority;
		END_IF
		req.pData := pData;
		req.nData := nData;
		req.deviceId := Client.ObjectInstance;
		stReq := ADR(req);
	END_IF
	
	IF pNull <> 0 AND_THEN pNull^ THEN
		req.nData := 0;
	ELSE
		req.nData := nData;
	END_IF
	
	IF SUPER^.Send() THEN
		IF pNull <> 0 THEN
			lastWriteValue.stCmdValue.bNull := pNull^;
			IF nData <= 4 THEN
				MEMCPY(ADR(lastWriteValue.stCmdValue.fValue), pData, nData);
			ELSIF lastWriteValue.nOther <> 0 THEN
				MEMCPY(lastWriteValue.nOther, pData, nData);
			END_IF
		ELSE
			IF nData <= 4 THEN
				MEMCPY(ADR(lastWriteValue.n32Value), pData, nData);
			ELSIF lastWriteValue.nOther <> 0 THEN
				MEMCPY(lastWriteValue.nOther, pData, nData);
			END_IF
		END_IF
		Send:=TRUE;
	END_IF
ELSE
	// (BETA) ... Output Error
END_IF
END_METHOD

METHOD PROTECTED OnError
VAR_INPUT
	eResult			: E_BACnetRM_Error;
	sLogCode		: STRING			:= '';
END_VAR
SUPER^.OnError(eResult, sLogCode);

IF fbWriteProp <> 0 THEN
	fbWriteProp^.Busy:=FALSE;
	fbWriteProp^.Error:=TRUE;
END_IF
END_METHOD

METHOD PROTECTED ProcessResult : HRESULT
VAR_INPUT
	pResult	: POINTER TO SendDataRequestResult;
END_VAR
bReady:=TRUE;

IF fbWriteProp <> 0 THEN
	fbWriteProp^.Busy:=FALSE;
	fbWriteProp^.Ready:=TRUE;
END_IF
END_METHOD

METHOD GetRequestType : E_BACnetRM_RequestType
VAR_INPUT
END_VAR
GetRequestType := E_BACnetRM_RequestType.eWrite;
END_METHOD

METHOD IsReady : BOOL
VAR_INPUT
END_VAR
VAR
	fValue : REAL;
END_VAR
IF SUPER^.IsReady() THEN
	IF pEnable = 0 OR_ELSE pEnable^ THEN
		IF fCOVIncrement <> 0.0 THEN
			MEMCPY(ADR(fValue), pData, SIZEOF(fValue));
			IF ABS(lastWriteValue.stCmdValue.fValue - fValue) > fCOVIncrement THEN
				IF pNull = 0 OR_ELSE NOT pNull^ THEN
					IsReady:=TRUE;
					RETURN;
				END_IF
			END_IF
			IF pNull <> 0 AND_THEN pNull^ <> lastWriteValue.stCmdValue.bNull THEN
				IsReady:=TRUE;
				RETURN;
			END_IF
		ELSE
			IF MEMCMP(ADR(lastWriteValue.n32Value), pData, nData) <> 0 THEN 
				IF pNull = 0 OR_ELSE NOT pNull^ THEN
					IsReady:=TRUE;
					RETURN;
				END_IF
			END_IF
			IF pNull <> 0 AND_THEN pNull^ <> lastWriteValue.stCmdValue.bNull THEN
				IsReady:=TRUE;
				RETURN;
			END_IF
		END_IF
	END_IF
END_IF
END_METHOD

END_FUNCTION_BLOCK

// POUs/Remote/Requests/FB_BACnetRM_WriteProperty
FUNCTION_BLOCK FB_BACnetRM_WriteProperty EXTENDS FB_BACnetRM_BaseProperty
VAR_INPUT CONSTANT
	{attribute 'initialize_on_call'}
	{attribute 'no_copy'}
	Device : REFERENCE TO FB_BACnet_Client;
	
	bRequestWPM : BOOL;
END_VAR

IF bExecuteOld <> bExecute AND NOT bBusy THEN
	IF NOT IsValid THEN
		bError:=TRUE;
		bReady:=FALSE;
	END_IF
	bExecuteOld := bExecute;
	Free();
	IF NOT Device.AddFifoWriteReq(THIS) THEN
		bError:=TRUE;
		bReady:=FALSE;
	ELSE
		bBusy:=TRUE;
		bError:=FALSE;
		bReady:=FALSE;
	END_IF
END_IF

METHOD PROTECTED OnExecuteChange : BOOL
OnExecuteChange := Device.AddFifoWriteReq(THIS);
END_METHOD

METHOD PROTECTED Free : BOOL
IF pRequest.pPtr <> 0 THEN
	IF bRequestWPM THEN
		__DELETE(pRequest.fbWpm);
	ELSE
		__DELETE(pRequest.fbWrite);
	END_IF
	pRequest.pPtr:=0;
END_IF
END_METHOD

METHOD FB_exit : BOOL
VAR_INPUT
	bInCopyCode : BOOL; // if TRUE, the exit method is called for exiting an instance that is copied afterwards (online change).
END_VAR
Free();
END_METHOD

PROPERTY IsValid : BOOL
GET
IsValid := __ISVALIDREF(Device);
END_GET
END_PROPERTY

END_FUNCTION_BLOCK

// POUs/Remote/Requests/[Internal]/FB_BACnetRM_ReqCov
{attribute 'c++_compatible'}
{attribute 'enable_dynamic_creation'}
{attribute 'hide'}
FUNCTION_BLOCK FB_BACnetRM_ReqCov EXTENDS FB_BACnetRM_ReqBasic
VAR_INPUT CONSTANT
	bConfirmed : BOOL;
	bUnsubscribed : BOOL;
	tLifetime : TIME := T#300S;
	fCOVIncrement : REAL := 0;
END_VAR
VAR_INPUT
	ePropID : E_BACnetPropIdentifier;
	pData : PVOID;
	nData : UDINT;
END_VAR
VAR_OUTPUT
	bSubsReady : BOOL;
END_VAR
VAR 
	req : SubscribeCovPropertyRequest;
	bSendSubs : BOOL := TRUE;
	pMaster : POINTER TO FB_BACnetRM_ReqCov;
	pCovSlaves : POINTER TO POINTER TO FB_BACnetRM_ReqCov;
	nCovSlaves : UDINT;
	nCovSlavesMax : UDINT;
END_VAR

IF NOT __ISVALIDREF(Client) THEN
	bError:=TRUE;
END_IF

SUPER^();

METHOD INTERNAL AddCovSlave : BOOL
VAR_INPUT
	pSlave : POINTER TO FB_BACnetRM_ReqCov;
END_VAR
VAR
	nTmp : UDINT;
	nTmpSize : UDINT;
	pTmp : POINTER TO POINTER TO FB_BACnetRM_ReqCov;
END_VAR
IF nCovSlaves+1 >= nCovSlavesMax THEN
	nTmp := nCovSlavesMax+10;
	nTmpSize := nTmp*SIZEOF(POINTER TO FB_BACnetRM_ReqCov);
	pTmp := __NEW(BYTE,nTmpSize);
	IF pTmp = 0 THEN
		RETURN;
	END_IF
	IF pCovSlaves <> 0 THEN
		MEMCPY(pTmp, pCovSlaves, nCovSlavesMax*SIZEOF(POINTER TO FB_BACnetRM_ReqCov));
		__DELETE(pCovSlaves);
	END_IF
	pCovSlaves:=pTmp;
	nCovSlavesMax:=nTmp;
END_IF

pCovSlaves[nCovSlaves]:=pSlave;
nCovSlaves:=nCovSlaves+1;
END_METHOD

{attribute 'hide'}
METHOD Send : BOOL
VAR
	iClientTmp : ITcIoBACnetPlcClient;
END_VAR
IF IsValid THEN
	IF NOT bSendSubs THEN
		RETURN;
	END_IF
	
	IF stReq = 0 THEN
		IF bUnsubscribed THEN
			req.issueConfirmedNotifications := FALSE;
			req.lifetime := 0;
			req.subscriberProcessIdentifier := 0;
		ELSE
			req.issueConfirmedNotifications := bConfirmed;
			req.lifetime := TIME_TO_DWORD(tLifetime) / 500;
			req.subscriberProcessIdentifier := 1;
		END_IF
		req.monitoredObjectIdentifier := iObject.ObjectID;
		req.covIncrement := fCOVIncrement;
		req.monitoredPropertyIdentifier.propertyIdentifier := ePropID;
		req.monitoredPropertyIdentifier.validFields := 1;	
	
		req.validFields := 2#0011111;
		IF req.covIncrement <> 0 THEN
			req.validFields := req.validFields +  2#100000;
		END_IF
	END_IF
	
	iClientTmp := Client.iClient;
	IF S_OK = iClientTmp.SendCOVSubscription(ADR(req), THIS^) THEN
		Send:=TRUE;
		StartTimer();
	END_IF
ELSE
	// (BETA) ... Output Error
END_IF
END_METHOD

METHOD PROTECTED ProcessResult : HRESULT
VAR_INPUT
	pResult	: POINTER TO SendDataRequestResult;
END_VAR
VAR
	pPropList : POINTER TO ST_BACnetRM_PropertyValueList;
	i : UDINT;
END_VAR
IF IsValid THEN
	IF pResult^.service = E_BACnetConfirmedService.SrvSubscribeCOV OR pResult^.service = E_BACnetConfirmedService.SrvSubscribeCOVProperty THEN
		bSubsReady:=TRUE;
		RETURN;
	END_IF
	
	IF pResult^.objectIdentifier = iObject.ObjectID THEN
		pPropList := pResult^.pData;
		WHILE pPropList <> 0 DO
			IF pPropList^.ePropID = ePropID THEN
				CopyRemoteData(iObject, ePropID, pData, nData, F_BACnet_EndOf(pPropList, SIZEOF(ST_BACnetRM_PropertyValueList)), pPropList^.nEntrySize AND 16#7FFFFFFF);
				bReady:=TRUE;
			END_IF
			pPropList := F_BACnet_NextListElem(pPropList, pPropList^.nEntrySize);
		END_WHILE
		bError := TRUE;
	END_IF
	
	IF pCovSlaves <> 0 AND nCovSlaves > 0 THEN
		FOR i:=0 TO nCovSlaves-1 DO
			pCovSlaves[i]^.ProcessResult(pResult);
		END_FOR
	END_IF
ELSE
	// (BETA) ... Output Error
END_IF
END_METHOD

METHOD PROTECTED StartTimer : BOOL
VAR_INPUT
END_VAR
timer(IN:=FALSE, PT:=tLifetime);
timer(IN:=TRUE, PT:=tLifetime);
END_METHOD

METHOD FB_Exit : BOOL
VAR_INPUT
	 bInCopyCode : BOOL; // if TRUE, the exit method is called for exiting an instance that is copied afterwards (online change).
END_VAR
VAR
	i : UDINT;
END_VAR
IF pCovSlaves <> 0 THEN
	__DELETE(pCovSlaves);
	pCovSlaves:=0;
END_IF
pMaster:=0;
END_METHOD

METHOD GetRequestType : E_BACnetRM_RequestType
VAR_INPUT
END_VAR
GetRequestType := E_BACnetRM_RequestType.eCov;
END_METHOD

METHOD IsReady : BOOL
VAR_INPUT
END_VAR
IF NOT bSendSubs THEN
	IsReady:=TRUE;
	RETURN;
END_IF

IsReady:=SUPER^.IsReady();
END_METHOD

PROPERTY Master : POINTER TO FB_BACnetRM_ReqCov
GET
Master:=pMaster;
END_GET
SET
pMaster:=Master;
END_SET
END_PROPERTY

PROPERTY SendSubscription : BOOL
GET
SendSubscription:=bSendSubs;
END_GET
SET
bSendSubs:=SendSubscription;
END_SET
END_PROPERTY

END_FUNCTION_BLOCK

// POUs/Remote/Objects/Basic/FB_BACnetRM_AV
FUNCTION_BLOCK FB_BACnetRM_AV EXTENDS FB_BACnetRM_EventObject
VAR_INPUT
	fPv 			: REAL;
	bEnablePv 		: BOOL;
	bNullPv 		: BOOL;	
END_VAR
VAR_INPUT CONSTANT PERSISTENT
	{region 'Fixed Parameters'}
		{attribute 'parameterCategory':='Value'}
		nPriority : BYTE := BACnet_Param.nRemotePrio_Default;
	{endregion}
END_VAR
VAR_OUTPUT
	fPresentValue 	: REAL;
END_VAR

SUPER^();

METHOD PROTECTED OnObjectStateChanged
SUPER^.OnObjectStateChanged();

SyncProperty(E_BACnetPropIdentifier.PropPresentValue, SIZEOF(fPresentValue), ADR(fPresentValue), E_BA_SyncModeRM.eRead);

SyncPropertyPrio(E_BACnetPropIdentifier.PropPresentValue, SIZEOF(fPv), ADR(fPv), ADR(bEnablePv), ADR(bNullPv), nPriority);
END_METHOD

METHOD FB_init : BOOL
VAR_INPUT
	bInitRetains : BOOL; // if TRUE, the retain variables are initialized (warm start / cold start)
	bInCopyCode : BOOL;  // if TRUE, the instance afterwards gets moved into the copy code (online change)
END_VAR
eObjectType := E_BACnetObjType.ObjAnalogValue;
END_METHOD

END_FUNCTION_BLOCK

// POUs/Remote/Objects/Basic/[Base]/FB_BACnetRM_EventObject
FUNCTION_BLOCK FB_BACnetRM_EventObject EXTENDS FB_BACnetRM_Object
VAR_OUTPUT
	bEvent						: BOOL;												// Indicates an active event
END_VAR
VAR
	{region 'Event'}
		stStateFlags			: ST_BA_StatusFlags;
	{endregion}
END_VAR

SUPER^();

bEvent := F_BA_IsDisturbed(stStateFlags);

METHOD PROTECTED OnObjectStateChanged
SUPER^.OnObjectStateChanged();

SyncProperty(E_BACnetPropIdentifier.PropStatusFlags, SIZEOF(stStateFlags), ADR(stStateFlags), E_BA_SyncModeRM.eRead);
END_METHOD

PROPERTY StateFlags : ST_BA_StatusFlags
GET
StateFlags := stStateFlags;
END_GET
END_PROPERTY

END_FUNCTION_BLOCK

// POUs/Remote/Objects/Basic/FB_BACnetRM_AV_Disp
FUNCTION_BLOCK FB_BACnetRM_AV_Disp EXTENDS FB_BACnetRM_Object
VAR_OUTPUT
	fPresentValue 	: REAL;
END_VAR

SUPER^();

METHOD PROTECTED OnObjectStateChanged
SUPER^.OnObjectStateChanged();

SyncProperty(E_BACnetPropIdentifier.PropPresentValue, SIZEOF(fPresentValue), ADR(fPresentValue), E_BA_SyncModeRM.eRead);
END_METHOD

METHOD FB_init : BOOL
VAR_INPUT
	bInitRetains : BOOL; // if TRUE, the retain variables are initialized (warm start / cold start)
	bInCopyCode : BOOL;  // if TRUE, the instance afterwards gets moved into the copy code (online change)
END_VAR
eObjectType := E_BACnetObjType.ObjAnalogValue;
END_METHOD

END_FUNCTION_BLOCK

// POUs/Remote/Objects/Basic/FB_BACnetRM_AV_Setp
FUNCTION_BLOCK FB_BACnetRM_AV_Setp EXTENDS FB_BACnetRM_Object
VAR_INPUT CONSTANT
	{region 'Operational Parameters'}
		{attribute 'parameterCategory':='Value'}
		fValue : REAL;
	{endregion}
END_VAR
VAR_OUTPUT
	fPresentValue 	: REAL;
END_VAR

SUPER^();

{attribute 'hide'}
METHOD OnCOV
VAR_INPUT
	ePropID		: E_BACnetPropIdentifier;
END_VAR
CASE (ePropID) OF
	E_BACnetPropIdentifier.PropPresentValue:
		fValue := fPresentValue;
		
ELSE
	SUPER^.OnCOV(ePropID);
END_CASE
END_METHOD

METHOD PROTECTED OnObjectStateChanged
SUPER^.OnObjectStateChanged();

SyncProperty(E_BACnetPropIdentifier.PropPresentValue, SIZEOF(fPresentValue), ADR(fPresentValue), E_BA_SyncModeRM.eRead);

SyncProperty(E_BACnetPropIdentifier.PropPresentValue, SIZEOF(fValue), ADR(fValue), E_BA_SyncModeRM.eWrite);
END_METHOD

METHOD FB_init : BOOL
VAR_INPUT
	bInitRetains : BOOL; // if TRUE, the retain variables are initialized (warm start / cold start)
	bInCopyCode : BOOL;  // if TRUE, the instance afterwards gets moved into the copy code (online change)
END_VAR
eObjectType := E_BACnetObjType.ObjAnalogValue;
END_METHOD

END_FUNCTION_BLOCK

// POUs/Remote/Objects/Basic/FB_BACnetRM_AI
FUNCTION_BLOCK FB_BACnetRM_AI EXTENDS FB_BACnetRM_EventObject
VAR_OUTPUT
	fPresentValue 	: REAL;
END_VAR

SUPER^();

METHOD PROTECTED OnObjectStateChanged
SUPER^.OnObjectStateChanged();

SyncProperty(E_BACnetPropIdentifier.PropPresentValue, SIZEOF(fPresentValue), ADR(fPresentValue), E_BA_SyncModeRM.eRead);
END_METHOD

METHOD FB_init : BOOL
VAR_INPUT
	bInitRetains : BOOL; // if TRUE, the retain variables are initialized (warm start / cold start)
	bInCopyCode : BOOL;  // if TRUE, the instance afterwards gets moved into the copy code (online change)
END_VAR
eObjectType := E_BACnetObjType.ObjAnalogInput;
END_METHOD

END_FUNCTION_BLOCK

// POUs/Remote/Objects/Basic/FB_BACnetRM_AO
FUNCTION_BLOCK FB_BACnetRM_AO EXTENDS FB_BACnetRM_EventObject
VAR_INPUT
	fPv 			: REAL;
	bEnablePv 		: BOOL;
	bNullPv 		: BOOL;
END_VAR
VAR_INPUT CONSTANT PERSISTENT
	{region 'Fixed Parameters'}
		{attribute 'parameterCategory':='Value'}
		nPriority : BYTE := BACnet_Param.nRemotePrio_Default;
	{endregion}
END_VAR
VAR_OUTPUT
	fPresentValue 	: REAL;
END_VAR

SUPER^();

METHOD PROTECTED OnObjectStateChanged
SUPER^.OnObjectStateChanged();

SyncProperty(E_BACnetPropIdentifier.PropPresentValue, SIZEOF(fPresentValue), ADR(fPresentValue), E_BA_SyncModeRM.eRead);

SyncPropertyPrio(E_BACnetPropIdentifier.PropPresentValue, SIZEOF(fPv), ADR(fPv), ADR(bEnablePv), ADR(bNullPv), nPriority);
END_METHOD

METHOD FB_init : BOOL
VAR_INPUT
	bInitRetains : BOOL; // if TRUE, the retain variables are initialized (warm start / cold start)
	bInCopyCode : BOOL;  // if TRUE, the instance afterwards gets moved into the copy code (online change)
END_VAR
eObjectType := E_BACnetObjType.ObjAnalogOutput;
END_METHOD

END_FUNCTION_BLOCK

// POUs/Remote/Objects/Basic/FB_BACnetRM_BV
FUNCTION_BLOCK FB_BACnetRM_BV EXTENDS FB_BACnetRM_EventObject
VAR_INPUT
	bPv 			: BOOL;
	bEnablePv 		: BOOL;
	bNullPv 		: BOOL;	
END_VAR
VAR_INPUT CONSTANT PERSISTENT
	{region 'Fixed Parameters'}
		{attribute 'parameterCategory':='Value'}
		nPriority : BYTE := BACnet_Param.nRemotePrio_Default;
	{endregion}
END_VAR
VAR_OUTPUT
	bPresentValue 	: BOOL;
END_VAR

SUPER^();

METHOD PROTECTED OnObjectStateChanged
SUPER^.OnObjectStateChanged();

SyncProperty(E_BACnetPropIdentifier.PropPresentValue, SIZEOF(bPresentValue), ADR(bPresentValue), E_BA_SyncModeRM.eRead);

SyncPropertyPrio(E_BACnetPropIdentifier.PropPresentValue, SIZEOF(bPv), ADR(bPv), ADR(bEnablePv), ADR(bNullPv), nPriority);
END_METHOD

METHOD FB_init : BOOL
VAR_INPUT
	bInitRetains : BOOL; // if TRUE, the retain variables are initialized (warm start / cold start)
	bInCopyCode : BOOL;  // if TRUE, the instance afterwards gets moved into the copy code (online change)
END_VAR
eObjectType := E_BACnetObjType.ObjBinaryValue;
END_METHOD

END_FUNCTION_BLOCK

// POUs/Remote/Objects/Basic/FB_BACnetRM_BV_Disp
FUNCTION_BLOCK FB_BACnetRM_BV_Disp EXTENDS FB_BACnetRM_Object
VAR_OUTPUT
	bPresentValue	: BOOL;
END_VAR

SUPER^();

METHOD PROTECTED OnObjectStateChanged
SUPER^.OnObjectStateChanged();

SyncProperty(E_BACnetPropIdentifier.PropPresentValue, SIZEOF(bPresentValue), ADR(bPresentValue), E_BA_SyncModeRM.eRead);
END_METHOD

METHOD FB_init : BOOL
VAR_INPUT
	bInitRetains : BOOL; // if TRUE, the retain variables are initialized (warm start / cold start)
	bInCopyCode : BOOL;  // if TRUE, the instance afterwards gets moved into the copy code (online change)
END_VAR
eObjectType := E_BACnetObjType.ObjBinaryValue;
END_METHOD

END_FUNCTION_BLOCK

// POUs/Remote/Objects/Basic/FB_BACnetRM_BV_Setp
FUNCTION_BLOCK FB_BACnetRM_BV_Setp EXTENDS FB_BACnetRM_Object
VAR_INPUT CONSTANT
	{region 'Operational Parameters'}
		{attribute 'parameterCategory':='Value'}
		bValue : BOOL;
	{endregion}
END_VAR
VAR_OUTPUT
	bPresentValue	: BOOL;
END_VAR

SUPER^();

{attribute 'hide'}
METHOD OnCOV
VAR_INPUT
	ePropID		: E_BACnetPropIdentifier;
END_VAR
CASE (ePropID) OF
	E_BACnetPropIdentifier.PropPresentValue:
		bValue := bPresentValue;
		
ELSE
	SUPER^.OnCOV(ePropID);
END_CASE
END_METHOD

METHOD PROTECTED OnObjectStateChanged
SUPER^.OnObjectStateChanged();

SyncProperty(E_BACnetPropIdentifier.PropPresentValue, SIZEOF(bPresentValue), ADR(bPresentValue), E_BA_SyncModeRM.eRead);

SyncProperty(E_BACnetPropIdentifier.PropPresentValue, SIZEOF(bValue), ADR(bValue), E_BA_SyncModeRM.eWrite);
END_METHOD

METHOD FB_init : BOOL
VAR_INPUT
	bInitRetains : BOOL; // if TRUE, the retain variables are initialized (warm start / cold start)
	bInCopyCode : BOOL;  // if TRUE, the instance afterwards gets moved into the copy code (online change)
END_VAR
eObjectType := E_BACnetObjType.ObjBinaryValue;
END_METHOD

END_FUNCTION_BLOCK

// POUs/Remote/Objects/Basic/FB_BACnetRM_BI
FUNCTION_BLOCK FB_BACnetRM_BI EXTENDS FB_BACnetRM_EventObject
VAR_OUTPUT
	bPresentValue 	: BOOL;
END_VAR

SUPER^();

METHOD PROTECTED OnObjectStateChanged
SUPER^.OnObjectStateChanged();

SyncProperty(E_BACnetPropIdentifier.PropPresentValue, SIZEOF(bPresentValue), ADR(bPresentValue), E_BA_SyncModeRM.eRead);
END_METHOD

METHOD FB_init : BOOL
VAR_INPUT
	bInitRetains : BOOL; // if TRUE, the retain variables are initialized (warm start / cold start)
	bInCopyCode : BOOL;  // if TRUE, the instance afterwards gets moved into the copy code (online change)
END_VAR
eObjectType := E_BACnetObjType.ObjBinaryInput;
END_METHOD

END_FUNCTION_BLOCK

// POUs/Remote/Objects/Basic/FB_BACnetRM_BO
FUNCTION_BLOCK FB_BACnetRM_BO EXTENDS FB_BACnetRM_EventObject
VAR_INPUT
	bPv 			: BOOL;
	bEnablePv 		: BOOL;
	bNullPv 		: BOOL;	
END_VAR
VAR_INPUT CONSTANT PERSISTENT
	{region 'Fixed Parameters'}
		{attribute 'parameterCategory':='Value'}
		nPriority : BYTE := BACnet_Param.nRemotePrio_Default;
	{endregion}
END_VAR
VAR_OUTPUT
	bPresentValue 	: BOOL;
END_VAR

SUPER^();

METHOD PROTECTED OnObjectStateChanged
SUPER^.OnObjectStateChanged();

SyncProperty(E_BACnetPropIdentifier.PropPresentValue, SIZEOF(bPresentValue), ADR(bPresentValue), E_BA_SyncModeRM.eRead);

SyncPropertyPrio(E_BACnetPropIdentifier.PropPresentValue, SIZEOF(bPv), ADR(bPv), ADR(bEnablePv), ADR(bNullPv), nPriority);
END_METHOD

METHOD FB_init : BOOL
VAR_INPUT
	bInitRetains : BOOL; // if TRUE, the retain variables are initialized (warm start / cold start)
	bInCopyCode : BOOL;  // if TRUE, the instance afterwards gets moved into the copy code (online change)
END_VAR
eObjectType := E_BACnetObjType.ObjBinaryOutput;
END_METHOD

END_FUNCTION_BLOCK

// POUs/Remote/Objects/Basic/FB_BACnetRM_MV
FUNCTION_BLOCK FB_BACnetRM_MV EXTENDS FB_BACnetRM_EventObject
VAR_INPUT
	nPv 			: UDINT;
	bEnablePv 		: BOOL;
	bNullPv 		: BOOL;	
END_VAR
VAR_INPUT CONSTANT PERSISTENT
	{region 'Fixed Parameters'}
		{attribute 'parameterCategory':='Value'}
		nPriority : BYTE := BACnet_Param.nRemotePrio_Default;
	{endregion}
END_VAR
VAR_OUTPUT
	nPresentValue 	: UDINT;
END_VAR

SUPER^();

METHOD PROTECTED OnObjectStateChanged
SUPER^.OnObjectStateChanged();

SyncProperty(E_BACnetPropIdentifier.PropPresentValue, SIZEOF(nPresentValue), ADR(nPresentValue), E_BA_SyncModeRM.eRead);

SyncPropertyPrio(E_BACnetPropIdentifier.PropPresentValue, SIZEOF(nPv), ADR(nPv), ADR(bEnablePv), ADR(bNullPv), nPriority);
END_METHOD

METHOD FB_init : BOOL
VAR_INPUT
	bInitRetains : BOOL; // if TRUE, the retain variables are initialized (warm start / cold start)
	bInCopyCode : BOOL;  // if TRUE, the instance afterwards gets moved into the copy code (online change)
END_VAR
eObjectType := E_BACnetObjType.ObjMultistateValue;
END_METHOD

END_FUNCTION_BLOCK

// POUs/Remote/Objects/Basic/FB_BACnetRM_MV_Disp
FUNCTION_BLOCK FB_BACnetRM_MV_Disp EXTENDS FB_BACnetRM_Object
VAR_OUTPUT
	nPresentValue		: UDINT		:= 1;
END_VAR

SUPER^();

METHOD PROTECTED OnObjectStateChanged
SUPER^.OnObjectStateChanged();

SyncProperty(E_BACnetPropIdentifier.PropPresentValue, SIZEOF(nPresentValue), ADR(nPresentValue), E_BA_SyncModeRM.eRead);
END_METHOD

METHOD FB_init : BOOL
VAR_INPUT
	bInitRetains : BOOL; // if TRUE, the retain variables are initialized (warm start / cold start)
	bInCopyCode : BOOL;  // if TRUE, the instance afterwards gets moved into the copy code (online change)
END_VAR
eObjectType := E_BACnetObjType.ObjMultistateValue;
END_METHOD

END_FUNCTION_BLOCK

// POUs/Remote/Objects/Basic/FB_BACnetRM_MV_Setp
FUNCTION_BLOCK FB_BACnetRM_MV_Setp EXTENDS FB_BACnetRM_Object
VAR_INPUT CONSTANT
	{region 'Operational Parameters'}
		{attribute 'parameterCategory':='Value'}
		nValue : UDINT;
	{endregion}
END_VAR
VAR_OUTPUT
	nPresentValue		: UDINT		:= 1;
END_VAR

SUPER^();

{attribute 'hide'}
METHOD OnCOV
VAR_INPUT
	ePropID		: E_BACnetPropIdentifier;
END_VAR
CASE (ePropID) OF
	E_BACnetPropIdentifier.PropPresentValue:
		nValue := nPresentValue;
		
ELSE
	SUPER^.OnCOV(ePropID);
END_CASE
END_METHOD

METHOD PROTECTED OnObjectStateChanged
SUPER^.OnObjectStateChanged();

SyncProperty(E_BACnetPropIdentifier.PropPresentValue, SIZEOF(nPresentValue), ADR(nPresentValue), E_BA_SyncModeRM.eRead);

SyncProperty(E_BACnetPropIdentifier.PropPresentValue, SIZEOF(nValue), ADR(nValue), E_BA_SyncModeRM.eWrite);
END_METHOD

METHOD FB_init : BOOL
VAR_INPUT
	bInitRetains : BOOL; // if TRUE, the retain variables are initialized (warm start / cold start)
	bInCopyCode : BOOL;  // if TRUE, the instance afterwards gets moved into the copy code (online change)
END_VAR
eObjectType := E_BACnetObjType.ObjMultistateValue;
END_METHOD

END_FUNCTION_BLOCK

// POUs/Remote/Objects/Basic/FB_BACnetRM_MI
FUNCTION_BLOCK FB_BACnetRM_MI EXTENDS FB_BACnetRM_EventObject
VAR_OUTPUT
	nPresentValue 	: UDINT;
END_VAR

SUPER^();

METHOD PROTECTED OnObjectStateChanged
SUPER^.OnObjectStateChanged();

SyncProperty(E_BACnetPropIdentifier.PropPresentValue, SIZEOF(nPresentValue), ADR(nPresentValue), E_BA_SyncModeRM.eRead);
END_METHOD

METHOD FB_init : BOOL
VAR_INPUT
	bInitRetains : BOOL; // if TRUE, the retain variables are initialized (warm start / cold start)
	bInCopyCode : BOOL;  // if TRUE, the instance afterwards gets moved into the copy code (online change)
END_VAR
eObjectType := E_BACnetObjType.ObjMultistateInput;
END_METHOD

END_FUNCTION_BLOCK

// POUs/Remote/Objects/Basic/FB_BACnetRM_MO
FUNCTION_BLOCK FB_BACnetRM_MO EXTENDS FB_BACnetRM_EventObject
VAR_INPUT
	nPv 			: UDINT;
	bEnablePv 		: BOOL;
	bNullPv 		: BOOL;	
END_VAR
VAR_INPUT CONSTANT PERSISTENT
	{region 'Fixed Parameters'}
		{attribute 'parameterCategory':='Value'}
		nPriority : BYTE := BACnet_Param.nRemotePrio_Default;
	{endregion}
END_VAR
VAR_OUTPUT
	nPresentValue 	: UDINT;
END_VAR

SUPER^();

METHOD PROTECTED OnObjectStateChanged
SUPER^.OnObjectStateChanged();

SyncProperty(E_BACnetPropIdentifier.PropPresentValue, SIZEOF(nPresentValue), ADR(nPresentValue), E_BA_SyncModeRM.eRead);

SyncPropertyPrio(E_BACnetPropIdentifier.PropPresentValue, SIZEOF(nPv), ADR(nPv), ADR(bEnablePv), ADR(bNullPv), nPriority);
END_METHOD

METHOD FB_init : BOOL
VAR_INPUT
	bInitRetains : BOOL; // if TRUE, the retain variables are initialized (warm start / cold start)
	bInCopyCode : BOOL;  // if TRUE, the instance afterwards gets moved into the copy code (online change)
END_VAR
eObjectType := E_BACnetObjType.ObjMultistateOutput;
END_METHOD

END_FUNCTION_BLOCK

// POUs/Remote/Objects/Basic/FB_BACnetRM_TLog
FUNCTION_BLOCK FB_BACnetRM_TLog EXTENDS FB_BACnetRM_BaseTLog

SUPER^();

METHOD FB_init : BOOL
VAR_INPUT
	bInitRetains : BOOL; // if TRUE, the retain variables are initialized (warm start / cold start)
	bInCopyCode : BOOL;  // if TRUE, the instance afterwards gets moved into the copy code (online change)
END_VAR
eObjectType := E_BACnetObjType.ObjTrendLog;
END_METHOD

END_FUNCTION_BLOCK

// POUs/Remote/Objects/Basic/[Base]/FB_BACnetRM_BaseTLog
FUNCTION_BLOCK FB_BACnetRM_BaseTLog EXTENDS FB_BACnetRM_EventObject
VAR_OUTPUT
	nRecordCount				: UDINT;
	nTotalRecordCount			: UDINT;
END_VAR

SUPER^();

METHOD PROTECTED OnObjectStateChanged
SUPER^.OnObjectStateChanged();

SyncProperty(E_BACnetPropIdentifier.PropRecordCount, SIZEOF(nRecordCount), ADR(nRecordCount), E_BA_SyncModeRM.eRead);
SyncProperty(E_BACnetPropIdentifier.PropTotalRecordCount, SIZEOF(nTotalRecordCount), ADR(nTotalRecordCount), E_BA_SyncModeRM.eRead);
END_METHOD

END_FUNCTION_BLOCK

// POUs/Remote/Objects/Basic/FB_BACnetRM_TLM
FUNCTION_BLOCK FB_BACnetRM_TLM EXTENDS FB_BACnetRM_BaseTLog

SUPER^();

METHOD FB_init : BOOL
VAR_INPUT
	bInitRetains : BOOL; // if TRUE, the retain variables are initialized (warm start / cold start)
	bInCopyCode : BOOL;  // if TRUE, the instance afterwards gets moved into the copy code (online change)
END_VAR
eObjectType := E_BACnetObjType.ObjTrendLogMultiple;
END_METHOD

END_FUNCTION_BLOCK

// POUs/Remote/Objects/Basic/FB_BACnetRM_Cal
FUNCTION_BLOCK FB_BACnetRM_Cal EXTENDS FB_BACnetRM_Object
VAR_OUTPUT
	bPresentValue 	: BOOL;
END_VAR

SUPER^();

METHOD PROTECTED OnObjectStateChanged
SUPER^.OnObjectStateChanged();

SyncProperty(E_BACnetPropIdentifier.PropPresentValue, SIZEOF(bPresentValue), ADR(bPresentValue), E_BA_SyncModeRM.eRead);
END_METHOD

METHOD FB_init : BOOL
VAR_INPUT
	bInitRetains : BOOL; // if TRUE, the retain variables are initialized (warm start / cold start)
	bInCopyCode : BOOL;  // if TRUE, the instance afterwards gets moved into the copy code (online change)
END_VAR
eObjectType := E_BACnetObjType.ObjCalendar;
END_METHOD

END_FUNCTION_BLOCK

// POUs/Remote/Objects/Basic/FB_BACnetRM_SchedA
FUNCTION_BLOCK FB_BACnetRM_SchedA EXTENDS FB_BACnetRM_Object
VAR_OUTPUT
	fPresentValue 	: REAL;
END_VAR

SUPER^();

METHOD PROTECTED OnObjectStateChanged
SUPER^.OnObjectStateChanged();

SyncProperty(E_BACnetPropIdentifier.PropPresentValue, SIZEOF(fPresentValue), ADR(fPresentValue), E_BA_SyncModeRM.eRead);
END_METHOD

METHOD FB_init : BOOL
VAR_INPUT
	bInitRetains : BOOL; // if TRUE, the retain variables are initialized (warm start / cold start)
	bInCopyCode : BOOL;  // if TRUE, the instance afterwards gets moved into the copy code (online change)
END_VAR
eObjectType := E_BACnetObjType.ObjSchedule;
END_METHOD

END_FUNCTION_BLOCK

// POUs/Remote/Objects/Basic/FB_BACnetRM_SchedB
FUNCTION_BLOCK FB_BACnetRM_SchedB EXTENDS FB_BACnetRM_Object
VAR_OUTPUT
	bPresentValue 	: BOOL;
END_VAR

SUPER^();

METHOD PROTECTED OnObjectStateChanged
SUPER^.OnObjectStateChanged();

SyncProperty(E_BACnetPropIdentifier.PropPresentValue, SIZEOF(bPresentValue), ADR(bPresentValue), E_BA_SyncModeRM.eRead);
END_METHOD

METHOD FB_init : BOOL
VAR_INPUT
	bInitRetains : BOOL; // if TRUE, the retain variables are initialized (warm start / cold start)
	bInCopyCode : BOOL;  // if TRUE, the instance afterwards gets moved into the copy code (online change)
END_VAR
eObjectType := E_BACnetObjType.ObjSchedule;
END_METHOD

END_FUNCTION_BLOCK

// POUs/Remote/Objects/Basic/FB_BACnetRM_SchedM
FUNCTION_BLOCK FB_BACnetRM_SchedM EXTENDS FB_BACnetRM_Object
VAR_OUTPUT
	nPresentValue 	: UDINT;
END_VAR

SUPER^();

METHOD PROTECTED OnObjectStateChanged
SUPER^.OnObjectStateChanged();

SyncProperty(E_BACnetPropIdentifier.PropPresentValue, SIZEOF(nPresentValue), ADR(nPresentValue), E_BA_SyncModeRM.eRead);
END_METHOD

METHOD FB_init : BOOL
VAR_INPUT
	bInitRetains : BOOL; // if TRUE, the retain variables are initialized (warm start / cold start)
	bInCopyCode : BOOL;  // if TRUE, the instance afterwards gets moved into the copy code (online change)
END_VAR
eObjectType := E_BACnetObjType.ObjSchedule;
END_METHOD

END_FUNCTION_BLOCK

// POUs/Remote/Objects/Basic/FB_BACnetRM_Loop
FUNCTION_BLOCK FB_BACnetRM_Loop EXTENDS FB_BACnetRM_EventObject
VAR_OUTPUT
	fPresentValue		: REAL;
	fSetpoint			: REAL;
	fCtrlVar			: REAL;
END_VAR

SUPER^();

METHOD PROTECTED OnObjectStateChanged
SUPER^.OnObjectStateChanged();

SyncProperty(E_BACnetPropIdentifier.PropPresentValue, SIZEOF(fPresentValue), ADR(fPresentValue), E_BA_SyncModeRM.eRead);
SyncProperty(E_BACnetPropIdentifier.PropSetpoint, SIZEOF(fSetpoint), ADR(fSetpoint), E_BA_SyncModeRM.eRead);
SyncProperty(E_BACnetPropIdentifier.PropControlledVariableValue, SIZEOF(fCtrlVar), ADR(fCtrlVar), E_BA_SyncModeRM.eRead);
END_METHOD

METHOD FB_init : BOOL
VAR_INPUT
	bInitRetains : BOOL; // if TRUE, the retain variables are initialized (warm start / cold start)
	bInCopyCode : BOOL;  // if TRUE, the instance afterwards gets moved into the copy code (online change)
END_VAR
eObjectType := E_BACnetObjType.ObjLoop;
END_METHOD

END_FUNCTION_BLOCK

// POUs/Remote/Objects/Convenience/FB_BACnetRM_CnvLoop
FUNCTION_BLOCK FB_BACnetRM_CnvLoop EXTENDS FB_BACnetRM_Loop
VAR_INPUT CONSTANT PERSISTENT
	{region 'Variable Parameters'}
		{attribute 'parameterCategory':='Config'}
		fPropertionalConstant : REAL;
		{attribute 'parameterCategory':='Config'}
		ePropertionalConstantUnit : E_BA_Unit;
		{attribute 'parameterCategory':='Config'}
		fIntegralConstant : REAL;
		{attribute 'parameterCategory':='Config'}
		eIntegralConstantUnit : E_BA_Unit;
		{attribute 'parameterCategory':='Config'}
		fDerivativeConstant : REAL;
		{attribute 'parameterCategory':='Config'}
		eDerivativeConstantUnit : E_BA_Unit;
	{endregion}
END_VAR

SUPER^();

METHOD PROTECTED OnObjectStateChanged
SUPER^.OnObjectStateChanged();

SyncProperty(E_BACnetPropIdentifier.PropProportionalConstant, SIZEOF(fPropertionalConstant), ADR(fPropertionalConstant), E_BA_SyncModeRM.eRead);
SyncProperty(E_BACnetPropIdentifier.PropProportionalConstantUnits, SIZEOF(ePropertionalConstantUnit), ADR(ePropertionalConstantUnit), E_BA_SyncModeRM.eRead);
SyncProperty(E_BACnetPropIdentifier.PropIntegralConstant, SIZEOF(fIntegralConstant), ADR(fIntegralConstant), E_BA_SyncModeRM.eRead);
SyncProperty(E_BACnetPropIdentifier.PropIntegralConstantUnits, SIZEOF(eIntegralConstantUnit), ADR(eIntegralConstantUnit), E_BA_SyncModeRM.eRead);
SyncProperty(E_BACnetPropIdentifier.PropDerivativeConstant, SIZEOF(fDerivativeConstant), ADR(fDerivativeConstant), E_BA_SyncModeRM.eRead);
SyncProperty(E_BACnetPropIdentifier.PropDerivativeConstantUnits, SIZEOF(eDerivativeConstantUnit), ADR(eDerivativeConstantUnit), E_BA_SyncModeRM.eRead);
END_METHOD

END_FUNCTION_BLOCK

// POUs/Remote/Objects/Basic/FB_BACnetRM_NC
FUNCTION_BLOCK FB_BACnetRM_NC EXTENDS FB_BACnetRM_Object
VAR_OUTPUT
	nNotificationClass		: UDINT;
END_VAR

SUPER^();

METHOD PROTECTED OnObjectStateChanged
SUPER^.OnObjectStateChanged();

SyncProperty(E_BACnetPropIdentifier.PropNotificationClass, SIZEOF(nNotificationClass), ADR(nNotificationClass), E_BA_SyncModeRM.eRead);
END_METHOD

METHOD FB_init : BOOL
VAR_INPUT
	bInitRetains : BOOL; // if TRUE, the retain variables are initialized (warm start / cold start)
	bInCopyCode : BOOL;  // if TRUE, the instance afterwards gets moved into the copy code (online change)
END_VAR
eObjectType := E_BACnetObjType.ObjNotificationClass;
END_METHOD

END_FUNCTION_BLOCK

// POUs/Remote/Objects/Basic/FB_BACnetRM_Acc
FUNCTION_BLOCK FB_BACnetRM_Acc EXTENDS FB_BACnetRM_EventObject
VAR_OUTPUT
	nPresentValue			: UDINT;
END_VAR

SUPER^();

METHOD PROTECTED OnObjectStateChanged
SUPER^.OnObjectStateChanged();

SyncProperty(E_BACnetPropIdentifier.PropPresentValue, SIZEOF(nPresentValue), ADR(nPresentValue), E_BA_SyncModeRM.eRead);
END_METHOD

METHOD FB_init : BOOL
VAR_INPUT
	bInitRetains : BOOL; // if TRUE, the retain variables are initialized (warm start / cold start)
	bInCopyCode : BOOL;  // if TRUE, the instance afterwards gets moved into the copy code (online change)
END_VAR
eObjectType := E_BACnetObjType.ObjAccumulator;
END_METHOD

END_FUNCTION_BLOCK

// POUs/Remote/Objects/Basic/FB_BACnetRM_PC
FUNCTION_BLOCK FB_BACnetRM_PC EXTENDS FB_BACnetRM_EventObject
VAR_OUTPUT
	fPresentValue			: REAL;
END_VAR

SUPER^();

METHOD PROTECTED OnObjectStateChanged
SUPER^.OnObjectStateChanged();

SyncProperty(E_BACnetPropIdentifier.PropPresentValue, SIZEOF(fPresentValue), ADR(fPresentValue), E_BA_SyncModeRM.eRead);
END_METHOD

METHOD FB_init : BOOL
VAR_INPUT
	bInitRetains : BOOL; // if TRUE, the retain variables are initialized (warm start / cold start)
	bInCopyCode : BOOL;  // if TRUE, the instance afterwards gets moved into the copy code (online change)
END_VAR
eObjectType := E_BACnetObjType.ObjPulseConverter;
END_METHOD

END_FUNCTION_BLOCK

// POUs/Remote/Objects/Basic/FB_BACnetRM_Prog
FUNCTION_BLOCK FB_BACnetRM_Prog EXTENDS FB_BACnetRM_EventObject
VAR_OUTPUT
	eState			: E_BACnet_ProgramState;
END_VAR

SUPER^();

METHOD PROTECTED OnObjectStateChanged
SUPER^.OnObjectStateChanged();

SyncProperty(E_BACnetPropIdentifier.PropProgramState, SIZEOF(eState), ADR(eState), E_BA_SyncModeRM.eRead);
END_METHOD

METHOD FB_init : BOOL
VAR_INPUT
	bInitRetains : BOOL; // if TRUE, the retain variables are initialized (warm start / cold start)
	bInCopyCode : BOOL;  // if TRUE, the instance afterwards gets moved into the copy code (online change)
END_VAR
eObjectType := E_BACnetObjType.ObjPulseConverter;
END_METHOD

END_FUNCTION_BLOCK

// POUs/Remote/Objects/Basic/FB_BACnetRM_Device
FUNCTION_BLOCK FB_BACnetRM_Device EXTENDS FB_BACnetRM_Object
VAR_OUTPUT
	bOperational		: BOOL;
END_VAR

IF (NOT bReady) THEN
	IF (nObjectInstance = 16#003FFFFF) THEN
		nObjectInstance:=Client.ObjectInstance;
	END_IF
END_IF

SUPER^();

METHOD PROTECTED OnObjectStateChanged
SUPER^.OnObjectStateChanged();

IF (nObjectInstance = 16#23FFFFF) THEN
	nObjectInstance := Client.ObjectInstance;
END_IF

SyncProperty(E_BACnetPropIdentifier.PropSystemStatus, SIZEOF(bOperational), ADR(bOperational), E_BA_SyncModeRM.eRead);
END_METHOD

METHOD FB_init : BOOL
VAR_INPUT
	bInitRetains : BOOL; // if TRUE, the retain variables are initialized (warm start / cold start)
	bInCopyCode : BOOL;  // if TRUE, the instance afterwards gets moved into the copy code (online change)
END_VAR
eObjectType := E_BACnetObjType.ObjDevice;
END_METHOD

END_FUNCTION_BLOCK

// POUs/Remote/Requests/[Internal]/FB_BACnetRM_ReqAckAlarm
{attribute 'c++_compatible'}
{attribute 'enable_dynamic_creation'}
{attribute 'hide'}
FUNCTION_BLOCK FB_BACnetRM_ReqAckAlarm EXTENDS FB_BACnetRM_ReqBase IMPLEMENTS ITcIoBACnetServiceResponseSink
VAR_INPUT
	sMsg : STRING;
	eAckEvent : E_BACnet_EventState;
END_VAR
VAR_OUTPUT
	bTsReady : BOOL;
	bReady : BOOL;
END_VAR
VAR
	req : AcknowledgeAlarmRequest;
	readTsReq : FB_BACnetRM_ReqRead;
	eventTs : ST_BACnet_EventTimeStamps;
END_VAR

IF NOT bTsReady THEN
	bTsReady := readTsReq.bReady;
END_IF

{attribute 'c++_compatible'}
{attribute 'minimal_input_size' := '4'}
{attribute 'pack_mode' := '4'}
{attribute 'hide'}
METHOD OnSendPropertyDataRequest : HRESULT
VAR_INPUT
	pResult	: POINTER TO SendDataRequestResult;
END_VAR
IF pResult <> 0 THEN
	IF F_BACnetRM_IsErrorSet(pResult) THEN
		bReady := FALSE;
		OnSendPropertyDataRequest:=S_FALSE;
	ELSE
		bReady := FALSE;	
	END_IF
END_IF
END_METHOD

{attribute 'hide'}
METHOD Send : BOOL
VAR
	_ClTmp : ITcIoBACnetPlcClient;
END_VAR
IF IsValid THEN
	req.acknowledgingProcessIdentifier := 0;
	req.eventObjectIdentifier := iObject.ObjectID;
	req.acknowledgmentSource := sMsg;
	req.eventStateAcknowledged := eAckEvent;
	IF eAckEvent = E_BACnet_EventState.eNormal THEN
		MEMCPY(ADR(req.timeStamp),ADR(eventTs.toNormal), SIZEOF(ST_BACnet_TimeStampDateTime));
	ELSIF eAckEvent = E_BACnet_EventState.eFault THEN
		MEMCPY(ADR(req.timeStamp),ADR(eventTs.toFault), SIZEOF(ST_BACnet_TimeStampDateTime));
	ELSE
		MEMCPY(ADR(req.timeStamp),ADR(eventTs.toOffNormal), SIZEOF(ST_BACnet_TimeStampDateTime));
	END_IF
	
	_ClTmp := Client.iClient;
	
	IF S_OK = _ClTmp.AcknowledgeAlarm(ADR(req), Client.ObjectInstance, THIS^) THEN
		Send:=TRUE;
	END_IF
ELSE
	// (BETA) ... Output Error
END_IF
END_METHOD

{attribute 'c++_compatible'}
{attribute 'minimal_input_size' := '4'}
{attribute 'pack_mode' := '4'}
{attribute 'hide'}
METHOD TcAddRef : UDINT
END_METHOD

{attribute 'c++_compatible'}
{attribute 'minimal_input_size' := '4'}
{attribute 'pack_mode' := '4'}
{attribute 'hide'}
METHOD TcQueryInterface : HRESULT
VAR_INPUT
	iid	: REFERENCE TO IID;
	pipItf	: POINTER TO PVOID;
END_VAR
VAR
	ipSink : ITcIoBACnetServiceResponseSink;
	ipUnknown : ITcUnknown;	
END_VAR
IF GuidsEqual(ADR(iid), ADR(TC_GLOBAL_IID_LIST.IID_ITcIoBACnetServiceResponseSink)) THEN
	ipSink := THIS^; // cast to interface pointer
	pipItf^ := ITCUNKNOWN_TO_PVOID(ipSink);
	TcAddRef();
	TcQueryInterface := S_OK;
ELSIF GuidsEqual(ADR(iid), ADR(TC_GLOBAL_IID_LIST.IID_ITcUnknown)) THEN
	ipUnknown := THIS^; // cast to interface pointer
	pipItf^ := ITCUNKNOWN_TO_PVOID(ipUnknown);
	TcAddRef();
	TcQueryInterface := S_OK;
ELSE
	TcQueryInterface := E_HRESULTAdsErr.NOINTERFACE ; //Call super if this fb extends some other
END_IF
END_METHOD

{attribute 'c++_compatible'}
{attribute 'minimal_input_size' := '4'}
{attribute 'pack_mode' := '4'}
{attribute 'hide'}
METHOD TcRelease : UDINT
END_METHOD

METHOD PRIVATE UpdateTimeStamp : BOOL
VAR_INPUT
END_VAR
IF IsValid THEN
	readTsReq(Client := Client, iObject:=iObject, ePropID:=E_BACnetPropIdentifier.PropEventTimeStamps, pData:=ADR(eventTs), nData:=SIZEOF(eventTs));
	readTsReq.Send();
ELSE
	// (BETA) ... Output Error
END_IF
END_METHOD

METHOD GetRequestType : E_BACnetRM_RequestType
VAR_INPUT
END_VAR
GetRequestType := E_BACnetRM_RequestType.eAcknowledge;
END_METHOD

METHOD IsReady : BOOL
VAR_INPUT
END_VAR
IsReady := bReady;
END_METHOD

END_FUNCTION_BLOCK

// POUs/Remote/Requests/[Internal]/FB_BACnetRM_ReqListAdd
{attribute 'c++_compatible'}
{attribute 'enable_dynamic_creation'}
{attribute 'hide'}
FUNCTION_BLOCK FB_BACnetRM_ReqListAdd EXTENDS FB_BACnetRM_ReqBasic
VAR_INPUT
	ePropID : E_BACnetPropIdentifier;
	pData : PVOID;
	nData : UDINT;
END_VAR
VAR 
	req : SendDataRequest;
END_VAR

IF NOT __ISVALIDREF(Client) THEN
	bError:=TRUE;
END_IF

SUPER^();

{attribute 'hide'}
METHOD Send : BOOL
IF IsValid THEN
	IF stReq = 0 THEN
		req.service := E_BACnetConfirmedService.SrvAddListElement;
		req.objectIdentifier := iObject.ObjectID;
		req.propertyIdentifier := ePropID;
		req.pData := pData;
		req.nData := nData;
		req.deviceId := Client.ObjectInstance;
		stReq := ADR(req);
	END_IF
	
	Send:=SUPER^.Send();
ELSE
	// (BETA) ... Output Error
END_IF
END_METHOD

METHOD PROTECTED ProcessResult : HRESULT
VAR_INPUT
	pResult	: POINTER TO SendDataRequestResult;
END_VAR
bReady:=TRUE;
END_METHOD

METHOD GetRequestType : E_BACnetRM_RequestType
VAR_INPUT
END_VAR
GetRequestType := E_BACnetRM_RequestType.eAddListElement;
END_METHOD

METHOD IsReady : BOOL
VAR_INPUT
END_VAR
IsReady := bReady;
END_METHOD

END_FUNCTION_BLOCK

// POUs/Remote/Requests/[Internal]/FB_BACnetRM_ReqListRem
{attribute 'c++_compatible'}
{attribute 'enable_dynamic_creation'}
{attribute 'hide'}
FUNCTION_BLOCK FB_BACnetRM_ReqListRem EXTENDS FB_BACnetRM_ReqBasic
VAR_INPUT
	ePropID : E_BACnetPropIdentifier;
	pData : PVOID;
	nData : UDINT;
END_VAR
VAR 
	req : SendDataRequest;
END_VAR

IF NOT __ISVALIDREF(Client) THEN
	bError:=TRUE;
END_IF

SUPER^();

{attribute 'hide'}
METHOD Send : BOOL
IF IsValid THEN
	IF stReq = 0 THEN
		req.service := E_BACnetConfirmedService.SrvRemoveListElement;
		req.objectIdentifier := iObject.ObjectID;
		req.propertyIdentifier := ePropID;
		req.pData := pData;
		req.nData := nData;
		req.deviceId := Client.ObjectInstance;
		stReq := ADR(req);
	END_IF
	
	Send:=SUPER^.Send();
ELSE
	// (BETA) ... Output Error
END_IF
END_METHOD

METHOD PROTECTED ProcessResult : HRESULT
VAR_INPUT
	pResult	: POINTER TO SendDataRequestResult;
END_VAR
bReady:=TRUE;
END_METHOD

METHOD GetRequestType : E_BACnetRM_RequestType
VAR_INPUT
END_VAR
GetRequestType := E_BACnetRM_RequestType.eRemoveListElement;
END_METHOD

END_FUNCTION_BLOCK

// TEST/TestPackage/Structure Samples/PRG02/TEMPLATES/Custom/H/HtgCirABC123/FB_BA_HtgCirABC123
FUNCTION_BLOCK FB_BA_HtgCirABC123 EXTENDS FB_BACnet_View
VAR_INPUT CONSTANT
	WthT							: FB_BACnet_AI_IO := (
										iParent 					:= THIS^,
										sObjectName					:= '\/WTHT',
										sDescription				:= '\/Aussentemperatur',
										sDeviceType					:= 'Temperatursensor',
										fResolution					:= 0.003051851,
										eUnit						:= E_BA_Unit.eTemperature_DegreesCelsius);
										
	FlWT							: FB_BACnet_AI_IO := (
										iParent 					:= THIS^,
										sObjectName					:= '\/TVL',
										sDescription				:= '\/Vorlauftemperatur',
										sDeviceType					:= 'Temperatursensor',
										fResolution					:= 0.003051851,
										eUnit						:= E_BA_Unit.eTemperature_DegreesCelsius);
	RtWT							: FB_BACnet_AI_IO := (
										iParent 					:= THIS^,
										sObjectName					:= '\/TRT',
										sDescription				:= '\/Rücklauftemperatur',
										sDeviceType					:= 'Temperatursensor',
										fResolution					:= 0.003051851,
										fScaleOffset				:= 0,
										eUnit						:= E_BA_Unit.eTemperature_DegreesCelsius);
										
	Sched							: FB_BACnet_SchedB := (
										iParent 					:= THIS^,
										sObjectName					:= '\/SCH01',
										sDescription				:= '\/Zeitschaltprogramm',
										tWeek						:= F_BACnet_SchedWeekly3xB(E_BA_Weekday.eMonday, E_BA_Weekday.eFriday, T#0H, FALSE, T#6H, TRUE, T#20H, FALSE));
										
	PID								: FB_BACnet_Loop := (
										iParent 					:= THIS^,
										sObjectName					:= '\/PID01',
										sDescription				:= '\/Vorlauftemperatirregler',
										eAction						:= E_BA_Action.eReverse,
										fPropertionalConstant		:= 1,
										fIntegralConstant			:= 180);	
										
	OpM								: FB_Bnet_H_OpM := (
										iParent 					:= THIS^);	
										
	SpG								: FB_Bnet_H_HtgCir_Sp := (
										iParent 					:= THIS^);	
										
	HtgLimit						: FB_Bnet_H_HtgCir_HtgLmt := (
										iParent 					:= THIS^);
										
	Vlv								: FB_Bnet_Vlv_013 := (
										iParent 					:= THIS^);	
										
	Pu								: FB_Bnet_Pu1st := (
										iParent 					:= THIS^);	
END_VAR
VAR // added by the converter: edge detectors and wires of the graphical bodies
    _w1 : ANY;
END_VAR

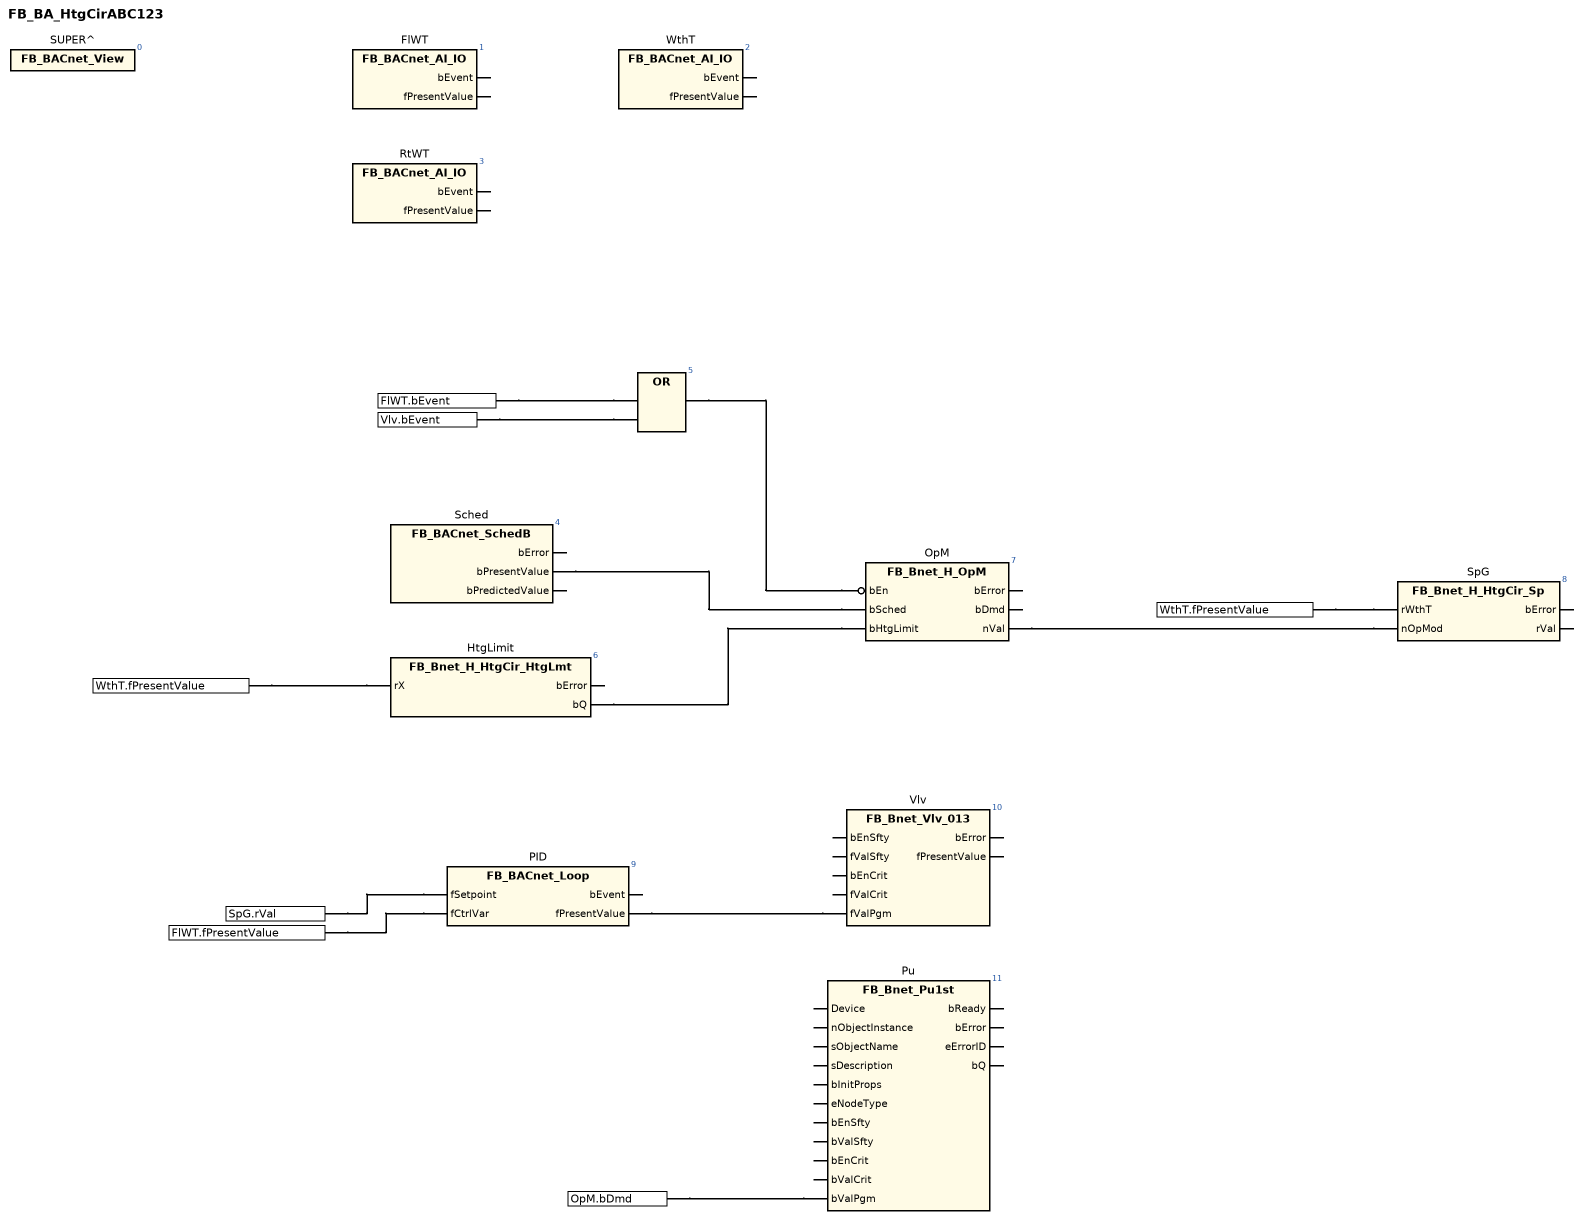
// note: 28 stored wires end on pins the file does not list and are not shown
SUPER^(); // FB_BACnet_View
FlWT(); // FB_BACnet_AI_IO
WthT(); // FB_BACnet_AI_IO
RtWT(); // FB_BACnet_AI_IO
Sched(); // FB_BACnet_SchedB
_w1 := FlWT.bEvent OR Vlv.bEvent;
HtgLimit(rX := WthT.fPresentValue); // FB_Bnet_H_HtgCir_HtgLmt
OpM(bEn := NOT _w1, bSched := Sched.bPresentValue, bHtgLimit := HtgLimit.bQ); // FB_Bnet_H_OpM
SpG(rWthT := WthT.fPresentValue, nOpMod := OpM.nVal); // FB_Bnet_H_HtgCir_Sp
PID(fSetpoint := SpG.rVal, fCtrlVar := FlWT.fPresentValue); // FB_BACnet_Loop
Vlv(fValPgm := PID.fPresentValue); // FB_Bnet_Vlv_013
Pu(bValPgm := OpM.bDmd); // FB_Bnet_Pu1st

METHOD FB_init : BOOL
VAR_INPUT
	bInitRetains : BOOL; // if TRUE, the retain variables are initialized (warm start / cold start)
	bInCopyCode : BOOL;  // if TRUE, the instance afterwards gets moved into the copy code (online change)
END_VAR
sObjectName		:= '\/HCR01';
sDescription	:= '\/Heizkreis';

Pu.BO.sObjectName := '\/XXXtest';
END_METHOD

END_FUNCTION_BLOCK

// TEST/TestPackage/TEMPLATES/HeatSupply/HeatingCircuit/FB_Bnet_H_HtgCir_HtgLmt
FUNCTION_BLOCK FB_Bnet_H_HtgCir_HtgLmt EXTENDS FB_BACnet_View
VAR_INPUT
	rX			: REAL;// Istwert	// Actual value
END_VAR
VAR_OUTPUT
	bQ			: BOOL;// Heizgrenzschalter Schaltbefehl Ein/Aus	// Heating limit switching command on/off
END_VAR
VAR
	Sp								:	FB_BACnet_AV_Setp := (
											iParent 			:= THIS^,
											sObjectName			:= '\/SP01',
											sDescription		:= '\/Sollwert',
											eUnit				:= E_BA_Unit.eTemperature_DegreesCelsius,
											fValue				:= 15.0);
											
	
	Hys				:	FB_Swi2P;//Hysterese Heizgrenze//Hysteresis heating limit
	
	Q								:	FB_BACnet_BV_Disp := (
											iParent 			:= THIS^,
											sObjectName			:= '\/STA01',
											sDescription		:= '\/Status',
											sActiveText			:= 'Ein',
											sInactiveText		:= 'Aus');
END_VAR
VAR // added by the converter: edge detectors and wires of the graphical bodies
    _w1, _w2 : ANY;
END_VAR

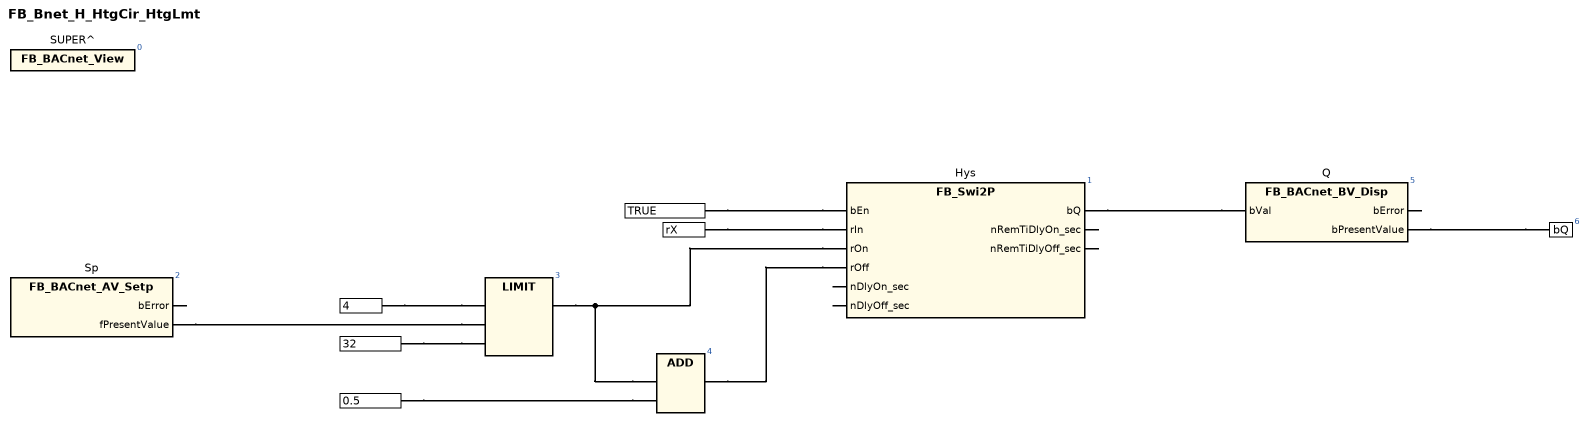
// note: 4 stored wires end on pins the file does not list and are not shown
SUPER^(); // FB_BACnet_View
Hys(bEn := TRUE, rIn := rX, rOn := _w1, rOff := _w2); // FB_Swi2P
Sp(); // FB_BACnet_AV_Setp
_w1 := LIMIT(4, Sp.fPresentValue, 32);
_w2 := _w1 + 0.5;
Q(bVal := Hys.bQ); // FB_BACnet_BV_Disp
bQ := Q.bPresentValue;

METHOD FB_init : BOOL
VAR_INPUT
	bInitRetains : BOOL; // if TRUE, the retain variables are initialized (warm start / cold start)
	bInCopyCode : BOOL;  // if TRUE, the instance afterwards gets moved into the copy code (online change)
END_VAR
sObjectName		:= '\/GW01';
sDescription	:= '\/Heizgrenzwert';
END_METHOD

END_FUNCTION_BLOCK

// TEST/TestPackage/TEMPLATES/HeatSupply/HeatingCircuit/FB_Swi2P
FUNCTION_BLOCK FB_Swi2P
VAR_INPUT
	bEn            : BOOL;// FB-enable
	rIn            : REAL;// input-value
	rOn            : REAL;// Switch-on point
	rOff           : REAL;// Switch-off point
	nDlyOn_sec		: UDINT;// (0..Const.nTiSec) switch-on delay [s]
	nDlyOff_sec		: UDINT;// (0..Const.nTiSec) switch-off delay [s]
END_VAR
VAR_OUTPUT
	bQ                 : BOOL;// control output
	nRemTiDlyOn_sec   : UDINT;// switch-on delay countdown [s]
	nRemTiDlyOff_sec  : UDINT;// switch-off delay countdown [s]
END_VAR
VAR
	tDlyOn				: TIME;
	tDlyOff				: TIME;
	tonDlyOn			: TON;
	tonDlyOff			: TON;
	rtrig				: R_TRIG;
	ftrig				: F_TRIG;
END_VAR

tDlyOn := TO_TIME(1000 * nDlyOn_sec);
tDlyOff := TO_TIME(1000 * nDlyOff_sec);

IF	bEn
THEN
	rtrig(CLK := rOn >= rOff);
	ftrig(CLK := rOn >= rOff);

	IF	rtrig.Q OR
		ftrig.Q
	THEN
		tonDlyOn(IN:= FALSE, PT:= T#0s);
		tonDlyOff(IN:= FALSE, PT:= T#0s);
		bQ := FALSE;
	END_IF

	IF	rOn >= rOff
	THEN
		IF	rOn = rOff
		THEN
			tonDlyOn(IN:= rIn >= rOn, PT:= tDlyOn);

			IF	tonDlyOn.Q
			THEN
				bQ := TRUE;
			END_IF

			tonDlyOff(IN:= bQ AND rIn < rOff, PT:= tDlyOff);

			IF	tonDlyOff.Q
			THEN
				bQ := FALSE;
			END_IF
		ELSE
			tonDlyOn(IN:= rIn >= rOn, PT:= tDlyOn);

			IF	tonDlyOn.Q
			THEN
				bQ := TRUE;
			END_IF

			tonDlyOff(IN:= bQ AND rIn <= rOff, PT:= tDlyOff);

			IF	tonDlyOff.Q
			THEN
				bQ := FALSE;
			END_IF
		END_IF
	ELSE
		tonDlyOn(IN:= rIn <= rOn, PT:= tDlyOn);

		IF	tonDlyOn.Q
		THEN
			bQ := TRUE;
		END_IF

		tonDlyOff(IN:= bQ AND rIn >= rOff, PT:= tDlyOff);

		IF	tonDlyOff.Q
		THEN
			bQ := FALSE;
		END_IF
	END_IF

	nRemTiDlyOn_sec := F_RemSecsTon(tonTimer := tonDlyOn);
	nRemTiDlyOff_sec := F_RemSecsTon(tonTimer := tonDlyOff);
ELSE
	tonDlyOn(IN:= FALSE, PT:= T#0s);
	tonDlyOff(IN:= FALSE, PT:= T#0s);
	nRemTiDlyOn_sec := nRemTiDlyOff_sec := 0;
	bQ := FALSE;
END_IF

END_FUNCTION_BLOCK

// TEST/TestPackage/TEMPLATES/Universal/AntiBlocking/F_RemSecsTon
{attribute 'hide'}
FUNCTION F_RemSecsTon : UDINT
VAR_INPUT
	tonTimer			: TON;		// Input of TON-Timer to be evaluated
END_VAR
VAR
	nRemTime_sec		: UDINT;		// remaining time in seconds of TP-Timeer
END_VAR

(*showing remaining Seconds of a timer
with +1-correction and 0, if timer is NOT running*)

nRemTime_sec	:= TO_UDINT((tonTimer.PT-tonTimer.ET)/1000)+1;

IF nRemTime_sec > TO_UDINT((tonTimer.PT)/1000) 		THEN
	nRemTime_sec := TO_UDINT((tonTimer.PT)/1000);
END_IF

IF tonTimer.Q		THEN
	nRemTime_sec := 0;
END_IF

F_RemSecsTon:=nRemTime_sec;

END_FUNCTION

// TEST/TestPackage/TEMPLATES/HeatSupply/FB_Bnet_H_OpM
FUNCTION_BLOCK FB_Bnet_H_OpM EXTENDS FB_BACnet_View
VAR_INPUT
	bEn				: BOOL;		//	Freigabe Betrieb							// Release operation
	bSched			: BOOL;		//	Zeitschaltplan Comfort und Economy Betrieb	// Switching schedule Comfort and Economy operation
	bHtgLimit		: BOOL;		// 	Heizgrenzschalter Schaltbefehl Ein/Aus		// Heating limit switching command on/off	
END_VAR
VAR_OUTPUT
	bDmd			: BOOL;		// 	Freigabe Heizkreis/Anforderung Wärmebedarf	// Enable heating circuit/requirement heat demand
	nVal			: UDINT;	// 	Betriebsart Protection,Economy,Comfort 		// Operating mode Protection,Economy,Comfort
END_VAR
VAR
	Man								:	FB_BACnet_MV_Setp := (
											iParent 			:= THIS^,
											sObjectName			:= '\/BAM01',
											sDescription		:= '\/Manuelle Betriebsart',
											sStateText			:= [ 'Auto', 'Schutzbetrieb', 'Economy', 'Comfort' ],
											nValue				:= 1);
											
	OpModPrioSwi				: FB_PrioSwi_UDI08;	//	Priorisierung Betriebsart	//	Prioritization operating mode

	PrOp							:	FB_BACnet_MV_Disp := (
											iParent 			:= THIS^,
											sObjectName			:= '\/BAS01',
											sDescription		:= '\/Aktuelle Betriebsart',
											sStateText			:= [ 'Schutzbetrieb', 'Economy', 'Comfort' ]);
											

	DmdPrioSwi					: FB_PrioSwi_B04;//Priorisierung Anforderung Wärmebedarf//Prioritization requirement heat demand

	Dmd								:	FB_BACnet_BV_Disp := (
											iParent 			:= THIS^,
											sObjectName			:= '\/AF01',
											sDescription		:= '\/Anforderung Heizen',
											sActiveText			:= 'Aktiv',
											sInactiveText		:= 'Inaktiv');
END_VAR
VAR // added by the converter: edge detectors and wires of the graphical bodies
    _w1, _w2, _w3, _w4, _w5, _w6 : ANY;
END_VAR

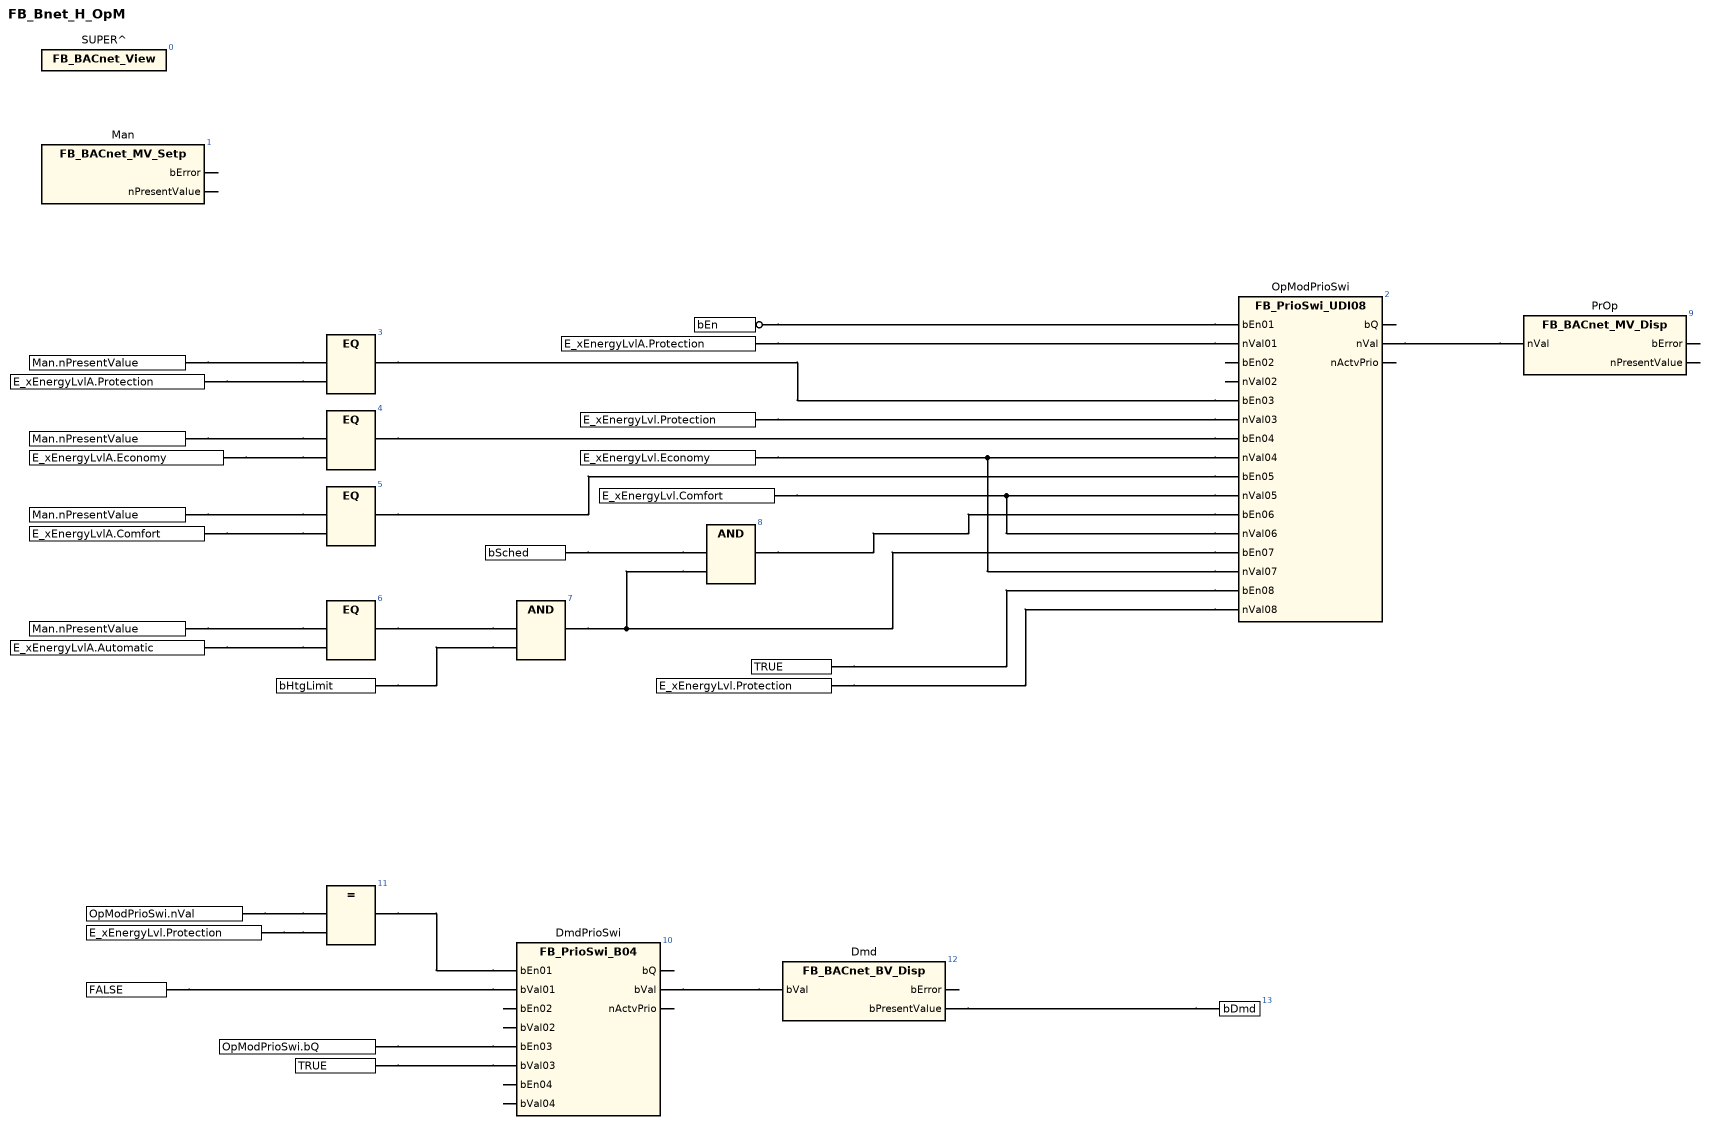
// note: 18 stored wires end on pins the file does not list and are not shown
SUPER^(); // FB_BACnet_View
Man(); // FB_BACnet_MV_Setp
OpModPrioSwi(
    bEn01 := NOT bEn,
    nVal01 := E_xEnergyLvlA.Protection,
    bEn03 := _w1,
    nVal03 := E_xEnergyLvl.Protection,
    bEn04 := _w2,
    nVal04 := E_xEnergyLvl.Economy,
    bEn05 := _w3,
    nVal05 := E_xEnergyLvl.Comfort,
    bEn06 := _w4,
    nVal06 := E_xEnergyLvl.Comfort,
    bEn07 := _w5,
    nVal07 := E_xEnergyLvl.Economy,
    bEn08 := TRUE,
    nVal08 := E_xEnergyLvl.Protection); // FB_PrioSwi_UDI08
_w1 := Man.nPresentValue = E_xEnergyLvlA.Protection;
_w2 := Man.nPresentValue = E_xEnergyLvlA.Economy;
_w3 := Man.nPresentValue = E_xEnergyLvlA.Comfort;
_w5 := Man.nPresentValue = E_xEnergyLvlA.Automatic AND bHtgLimit;
_w4 := bSched AND _w5;
PrOp(nVal := OpModPrioSwi.nVal); // FB_BACnet_MV_Disp
DmdPrioSwi(bEn01 := _w6, bVal01 := FALSE, bEn03 := OpModPrioSwi.bQ, bVal03 := TRUE); // FB_PrioSwi_B04
_w6 := OpModPrioSwi.nVal = E_xEnergyLvl.Protection;
Dmd(bVal := DmdPrioSwi.bVal); // FB_BACnet_BV_Disp
bDmd := Dmd.bPresentValue;

METHOD FB_init : BOOL
VAR_INPUT
	bInitRetains : BOOL; // if TRUE, the retain variables are initialized (warm start / cold start)
	bInCopyCode : BOOL;  // if TRUE, the instance afterwards gets moved into the copy code (online change)
END_VAR
sObjectName		:= '\/OPM01';
sDescription	:= '\/Betriebsart';
END_METHOD

END_FUNCTION_BLOCK

// TEST/TestPackage/TEMPLATES/HeatSupply/FB_PrioSwi_UDI08
FUNCTION_BLOCK FB_PrioSwi_UDI08
VAR_INPUT
	bEn01		: BOOL;		// Enabling the priority value
	nVal01		: UDINT;	// Priority value
	bEn02		: BOOL;		// Enabling the priority value
	nVal02		: UDINT;	// Priority value
	bEn03		: BOOL;		// Enabling the priority value
	nVal03		: UDINT;	// Priority value
	bEn04		: BOOL;		// Enabling the priority value
	nVal04		: UDINT;	// Priority value
	bEn05		: BOOL;		// Enabling the priority value
	nVal05		: UDINT;	// Priority value
	bEn06		: BOOL;		// Enabling the priority value
	nVal06		: UDINT;	// Priority value
	bEn07		: BOOL;		// Enabling the priority value
	nVal07		: UDINT;	// Priority value
	bEn08		: BOOL;		// Enabling the priority value
	nVal08		: UDINT;	// Priority value
END_VAR
VAR_OUTPUT
	bQ			: BOOL;		// Output to indicate whether a priority is enabled
	nVal		: UDINT;	// Output of the value of the current (highest) priority that is enabled
	nActvPrio	: UDINT;		// Current (highest) priority that is enabled
END_VAR
VAR
	arrEn		: ARRAY [1..cBA_PrioSwiUDI08] OF BOOL;
	arrVal		: ARRAY [1..cBA_PrioSwiUDI08] OF UDINT;
	i			: UDINT;
END_VAR
VAR CONSTANT
	cBA_PrioSwiUDI08    : UDINT := 8;
END_VAR

arrEn[1] := bEn01;
arrEn[2] := bEn02;
arrEn[3] := bEn03;
arrEn[4] := bEn04;
arrEn[5] := bEn05;
arrEn[6] := bEn06;
arrEn[7] := bEn07;
arrEn[8] := bEn08;

arrVal[1] := nVal01;
arrVal[2] := nVal02;
arrVal[3] := nVal03;
arrVal[4] := nVal04;
arrVal[5] := nVal05;
arrVal[6] := nVal06;
arrVal[7] := nVal07;
arrVal[8] := nVal08;

bQ := FALSE;
nVal := 0;
nActvPrio := Const.nNoActvPrio;

FOR i := 1 TO cBA_PrioSwiUDI08 BY 1 DO
	IF	arrEn[i] = TRUE
	THEN
		bQ := TRUE;
		nVal := arrVal[i];
		nActvPrio := i;
		EXIT;
	END_IF
END_FOR

END_FUNCTION_BLOCK

// TEST/TestPackage/TEMPLATES/HeatSupply/FB_PrioSwi_B04
FUNCTION_BLOCK FB_PrioSwi_B04
VAR_INPUT
	bEn01		: BOOL;	// Enabling the priority value
	bVal01		: BOOL;	// Priority value
	bEn02		: BOOL;	// Enabling the priority value
	bVal02		: BOOL;	// Priority value
	bEn03		: BOOL;	// Enabling the priority value
	bVal03		: BOOL;	// Priority value
	bEn04		: BOOL;	// Enabling the priority value
	bVal04		: BOOL;	// Priority value
END_VAR
VAR_OUTPUT
	bQ			: BOOL;	// Output to indicate whether a priority is enabled
	bVal		: BOOL;	// Output of the value of the current (highest) priority that is enabled
	nActvPrio	: UDINT;	// Current (highest) priority that is enabled
END_VAR
VAR
	arrEn		: ARRAY [1..cBA_PrioSwiB04] OF BOOL;
	arrVal		: ARRAY [1..cBA_PrioSwiB04] OF BOOL;
	i			: UDINT;
END_VAR
VAR CONSTANT
	cBA_PrioSwiB04    : UDINT := 4;
END_VAR

